(* Logix 5000 project; controller reports 1756-L63 rev 20.11; software revision 20.04; part 17 of 52 *)

        [888].time.Minute := 24, [888].time.Second := 59, [889].log_data[0].min := 1.0, [889].log_data[0].max := 1.0, [889].log_data[0].total := 300.0, [889].log_data[0].time := 300.0, [889].log_data[0].minminute := 25, [889].log_data[0].maxminute := 25, [889].log_data[0].valid := 1, [889].log_data[1].valid := 1, [889].log_data[2].valid := 1, [889].log_data[3].valid := 1, [889].log_data[4].valid := 1, [889].log_data[5].valid := 1, [889].log_data[6].valid := 1, [889].log_data[7].valid := 1, [889].log_data[8].valid := 1, [889].log_data[9].valid := 1, [889].log_data[10].valid := 1, [889].log_data[11].valid := 1, [889].log_data[12].valid := 1, [889].log_data[13].valid := 1, [889].log_data[14].valid := 1, [889].log_data[15].valid := 1, [889].log_data[16].valid := 1, [889].log_data[17].valid := 1, [889].log_data[18].valid := 1, [889].log_data[19].valid := 1, [889].time.Year := 2023, [889].time.Month := 1, [889].time.Day := 12, [889].time.Hour := 18, [889].time.Minute := 29, [889].time.Second := 59, [890].log_data[0].min := 1.0, [890].log_data[0].max := 1.0, [890].log_data[0].total := 300.0, [890].log_data[0].time := 300.0, [890].log_data[0].minminute := 30, [890].log_data[0].maxminute := 30, [890].log_data[0].valid := 1, [890].log_data[1].valid := 1, [890].log_data[2].valid := 1, [890].log_data[3].valid := 1, [890].log_data[4].valid := 1, [890].log_data[5].valid := 1, [890].log_data[6].valid := 1, [890].log_data[7].valid := 1, [890].log_data[8].valid := 1, [890].log_data[9].valid := 1, [890].log_data[10].valid := 1, [890].log_data[11].valid := 1, [890].log_data[12].valid := 1, [890].log_data[13].valid := 1, [890].log_data[14].valid := 1, [890].log_data[15].valid := 1, [890].log_data[16].valid := 1, [890].log_data[17].valid := 1, [890].log_data[18].valid := 1, [890].log_data[19].valid := 1,
        [890].time.Year := 2023, [890].time.Month := 1, [890].time.Day := 12, [890].time.Hour := 18, [890].time.Minute := 34, [890].time.Second := 59, [891].log_data[0].min := 1.0, [891].log_data[0].max := 1.0, [891].log_data[0].total := 300.0, [891].log_data[0].time := 300.0, [891].log_data[0].minminute := 35, [891].log_data[0].maxminute := 35, [891].log_data[0].valid := 1, [891].log_data[1].valid := 1, [891].log_data[2].valid := 1, [891].log_data[3].valid := 1, [891].log_data[4].valid := 1, [891].log_data[5].valid := 1, [891].log_data[6].valid := 1, [891].log_data[7].valid := 1, [891].log_data[8].valid := 1, [891].log_data[9].valid := 1, [891].log_data[10].valid := 1, [891].log_data[11].valid := 1, [891].log_data[12].valid := 1, [891].log_data[13].valid := 1, [891].log_data[14].valid := 1, [891].log_data[15].valid := 1, [891].log_data[16].valid := 1, [891].log_data[17].valid := 1, [891].log_data[18].valid := 1, [891].log_data[19].valid := 1, [891].time.Year := 2023, [891].time.Month := 1, [891].time.Day := 12, [891].time.Hour := 18, [891].time.Minute := 39, [891].time.Second := 59, [892].log_data[0].min := 1.0, [892].log_data[0].max := 1.0, [892].log_data[0].total := 300.0, [892].log_data[0].time := 300.0, [892].log_data[0].minminute := 40, [892].log_data[0].maxminute := 40, [892].log_data[0].valid := 1, [892].log_data[1].valid := 1, [892].log_data[2].valid := 1, [892].log_data[3].valid := 1, [892].log_data[4].valid := 1, [892].log_data[5].valid := 1, [892].log_data[6].valid := 1, [892].log_data[7].valid := 1, [892].log_data[8].valid := 1, [892].log_data[9].valid := 1, [892].log_data[10].valid := 1, [892].log_data[11].valid := 1, [892].log_data[12].valid := 1, [892].log_data[13].valid := 1, [892].log_data[14].valid := 1, [892].log_data[15].valid := 1,
        [892].log_data[16].valid := 1, [892].log_data[17].valid := 1, [892].log_data[18].valid := 1, [892].log_data[19].valid := 1, [892].time.Year := 2023, [892].time.Month := 1, [892].time.Day := 12, [892].time.Hour := 18, [892].time.Minute := 44, [892].time.Second := 59, [893].log_data[0].min := 1.0, [893].log_data[0].max := 1.0, [893].log_data[0].total := 300.0, [893].log_data[0].time := 300.0, [893].log_data[0].minminute := 45, [893].log_data[0].maxminute := 45, [893].log_data[0].valid := 1, [893].log_data[1].valid := 1, [893].log_data[2].valid := 1, [893].log_data[3].valid := 1, [893].log_data[4].valid := 1, [893].log_data[5].valid := 1, [893].log_data[6].valid := 1, [893].log_data[7].valid := 1, [893].log_data[8].valid := 1, [893].log_data[9].valid := 1, [893].log_data[10].valid := 1, [893].log_data[11].valid := 1, [893].log_data[12].valid := 1, [893].log_data[13].valid := 1, [893].log_data[14].valid := 1, [893].log_data[15].valid := 1, [893].log_data[16].valid := 1, [893].log_data[17].valid := 1, [893].log_data[18].valid := 1, [893].log_data[19].valid := 1, [893].time.Year := 2023, [893].time.Month := 1, [893].time.Day := 12, [893].time.Hour := 18, [893].time.Minute := 49, [893].time.Second := 59, [894].log_data[0].min := 1.0, [894].log_data[0].max := 1.0, [894].log_data[0].total := 300.0, [894].log_data[0].time := 300.0, [894].log_data[0].minminute := 50, [894].log_data[0].maxminute := 50, [894].log_data[0].valid := 1, [894].log_data[1].valid := 1, [894].log_data[2].valid := 1, [894].log_data[3].valid := 1, [894].log_data[4].valid := 1, [894].log_data[5].valid := 1, [894].log_data[6].valid := 1, [894].log_data[7].valid := 1, [894].log_data[8].valid := 1, [894].log_data[9].valid := 1, [894].log_data[10].valid := 1, [894].log_data[11].valid := 1,
        [894].log_data[12].valid := 1, [894].log_data[13].valid := 1, [894].log_data[14].valid := 1, [894].log_data[15].valid := 1, [894].log_data[16].valid := 1, [894].log_data[17].valid := 1, [894].log_data[18].valid := 1, [894].log_data[19].valid := 1, [894].time.Year := 2023, [894].time.Month := 1, [894].time.Day := 12, [894].time.Hour := 18, [894].time.Minute := 54, [894].time.Second := 59, [895].log_data[0].min := 1.0, [895].log_data[0].max := 1.0, [895].log_data[0].total := 300.0, [895].log_data[0].time := 300.0, [895].log_data[0].minminute := 55, [895].log_data[0].maxminute := 55, [895].log_data[0].valid := 1, [895].log_data[1].valid := 1, [895].log_data[2].valid := 1, [895].log_data[3].valid := 1, [895].log_data[4].valid := 1, [895].log_data[5].valid := 1, [895].log_data[6].valid := 1, [895].log_data[7].valid := 1, [895].log_data[8].valid := 1, [895].log_data[9].valid := 1, [895].log_data[10].valid := 1, [895].log_data[11].valid := 1, [895].log_data[12].valid := 1, [895].log_data[13].valid := 1, [895].log_data[14].valid := 1, [895].log_data[15].valid := 1, [895].log_data[16].valid := 1, [895].log_data[17].valid := 1, [895].log_data[18].valid := 1, [895].log_data[19].valid := 1, [895].time.Year := 2023, [895].time.Month := 1, [895].time.Day := 12, [895].time.Hour := 18, [895].time.Minute := 59, [895].time.Second := 59, [896].log_data[0].min := 1.0, [896].log_data[0].max := 1.0, [896].log_data[0].total := 300.0, [896].log_data[0].time := 300.0, [896].log_data[0].valid := 1, [896].log_data[1].valid := 1, [896].log_data[2].valid := 1, [896].log_data[3].valid := 1, [896].log_data[4].valid := 1, [896].log_data[5].valid := 1, [896].log_data[6].valid := 1, [896].log_data[7].valid := 1, [896].log_data[8].valid := 1, [896].log_data[9].valid := 1,
        [896].log_data[10].valid := 1, [896].log_data[11].valid := 1, [896].log_data[12].valid := 1, [896].log_data[13].valid := 1, [896].log_data[14].valid := 1, [896].log_data[15].valid := 1, [896].log_data[16].valid := 1, [896].log_data[17].valid := 1, [896].log_data[18].valid := 1, [896].log_data[19].valid := 1, [896].time.Year := 2023, [896].time.Month := 1, [896].time.Day := 12, [896].time.Hour := 19, [896].time.Minute := 4, [896].time.Second := 59, [897].log_data[0].min := 1.0, [897].log_data[0].max := 1.0, [897].log_data[0].total := 300.0, [897].log_data[0].time := 300.0, [897].log_data[0].minminute := 5, [897].log_data[0].maxminute := 5, [897].log_data[0].valid := 1, [897].log_data[1].valid := 1, [897].log_data[2].valid := 1, [897].log_data[3].valid := 1, [897].log_data[4].valid := 1, [897].log_data[5].valid := 1, [897].log_data[6].valid := 1, [897].log_data[7].valid := 1, [897].log_data[8].valid := 1, [897].log_data[9].valid := 1, [897].log_data[10].valid := 1, [897].log_data[11].valid := 1, [897].log_data[12].valid := 1, [897].log_data[13].valid := 1, [897].log_data[14].valid := 1, [897].log_data[15].valid := 1, [897].log_data[16].valid := 1, [897].log_data[17].valid := 1, [897].log_data[18].valid := 1, [897].log_data[19].valid := 1, [897].time.Year := 2023, [897].time.Month := 1, [897].time.Day := 12, [897].time.Hour := 19, [897].time.Minute := 9, [897].time.Second := 59, [898].log_data[0].min := 1.0, [898].log_data[0].max := 1.0, [898].log_data[0].total := 300.0, [898].log_data[0].time := 300.0, [898].log_data[0].minminute := 10, [898].log_data[0].maxminute := 10, [898].log_data[0].valid := 1, [898].log_data[1].valid := 1, [898].log_data[2].valid := 1, [898].log_data[3].valid := 1, [898].log_data[4].valid := 1, [898].log_data[5].valid := 1,
        [898].log_data[6].valid := 1, [898].log_data[7].valid := 1, [898].log_data[8].valid := 1, [898].log_data[9].valid := 1, [898].log_data[10].valid := 1, [898].log_data[11].valid := 1, [898].log_data[12].valid := 1, [898].log_data[13].valid := 1, [898].log_data[14].valid := 1, [898].log_data[15].valid := 1, [898].log_data[16].valid := 1, [898].log_data[17].valid := 1, [898].log_data[18].valid := 1, [898].log_data[19].valid := 1, [898].time.Year := 2023, [898].time.Month := 1, [898].time.Day := 12, [898].time.Hour := 19, [898].time.Minute := 14, [898].time.Second := 59, [899].log_data[0].min := 1.0, [899].log_data[0].max := 1.0, [899].log_data[0].total := 300.0, [899].log_data[0].time := 300.0, [899].log_data[0].minminute := 15, [899].log_data[0].maxminute := 15, [899].log_data[0].valid := 1, [899].log_data[1].valid := 1, [899].log_data[2].valid := 1, [899].log_data[3].valid := 1, [899].log_data[4].valid := 1, [899].log_data[5].valid := 1, [899].log_data[6].valid := 1, [899].log_data[7].valid := 1, [899].log_data[8].valid := 1, [899].log_data[9].valid := 1, [899].log_data[10].valid := 1, [899].log_data[11].valid := 1, [899].log_data[12].valid := 1, [899].log_data[13].valid := 1, [899].log_data[14].valid := 1, [899].log_data[15].valid := 1, [899].log_data[16].valid := 1, [899].log_data[17].valid := 1, [899].log_data[18].valid := 1, [899].log_data[19].valid := 1, [899].time.Year := 2023, [899].time.Month := 1, [899].time.Day := 12, [899].time.Hour := 19, [899].time.Minute := 19, [899].time.Second := 59, [900].log_data[0].min := 1.0, [900].log_data[0].max := 1.0, [900].log_data[0].total := 300.0, [900].log_data[0].time := 300.0, [900].log_data[0].minminute := 20, [900].log_data[0].maxminute := 20, [900].log_data[0].valid := 1, [900].log_data[1].valid := 1,
        [900].log_data[2].valid := 1, [900].log_data[3].valid := 1, [900].log_data[4].valid := 1, [900].log_data[5].valid := 1, [900].log_data[6].valid := 1, [900].log_data[7].valid := 1, [900].log_data[8].valid := 1, [900].log_data[9].valid := 1, [900].log_data[10].valid := 1, [900].log_data[11].valid := 1, [900].log_data[12].valid := 1, [900].log_data[13].valid := 1, [900].log_data[14].valid := 1, [900].log_data[15].valid := 1, [900].log_data[16].valid := 1, [900].log_data[17].valid := 1, [900].log_data[18].valid := 1, [900].log_data[19].valid := 1, [900].time.Year := 2023, [900].time.Month := 1, [900].time.Day := 12, [900].time.Hour := 19, [900].time.Minute := 24, [900].time.Second := 59, [901].log_data[0].min := 1.0, [901].log_data[0].max := 1.0, [901].log_data[0].total := 300.0, [901].log_data[0].time := 300.0, [901].log_data[0].minminute := 25, [901].log_data[0].maxminute := 25, [901].log_data[0].valid := 1, [901].log_data[1].valid := 1, [901].log_data[2].valid := 1, [901].log_data[3].valid := 1, [901].log_data[4].valid := 1, [901].log_data[5].valid := 1, [901].log_data[6].valid := 1, [901].log_data[7].valid := 1, [901].log_data[8].valid := 1, [901].log_data[9].valid := 1, [901].log_data[10].valid := 1, [901].log_data[11].valid := 1, [901].log_data[12].valid := 1, [901].log_data[13].valid := 1, [901].log_data[14].valid := 1, [901].log_data[15].valid := 1, [901].log_data[16].valid := 1, [901].log_data[17].valid := 1, [901].log_data[18].valid := 1, [901].log_data[19].valid := 1, [901].time.Year := 2023, [901].time.Month := 1, [901].time.Day := 12, [901].time.Hour := 19, [901].time.Minute := 29, [901].time.Second := 59, [902].log_data[0].min := 1.0, [902].log_data[0].max := 1.0, [902].log_data[0].total := 300.0, [902].log_data[0].time := 300.0,
        [902].log_data[0].minminute := 30, [902].log_data[0].maxminute := 30, [902].log_data[0].valid := 1, [902].log_data[1].valid := 1, [902].log_data[2].valid := 1, [902].log_data[3].valid := 1, [902].log_data[4].valid := 1, [902].log_data[5].valid := 1, [902].log_data[6].valid := 1, [902].log_data[7].valid := 1, [902].log_data[8].valid := 1, [902].log_data[9].valid := 1, [902].log_data[10].valid := 1, [902].log_data[11].valid := 1, [902].log_data[12].valid := 1, [902].log_data[13].valid := 1, [902].log_data[14].valid := 1, [902].log_data[15].valid := 1, [902].log_data[16].valid := 1, [902].log_data[17].valid := 1, [902].log_data[18].valid := 1, [902].log_data[19].valid := 1, [902].time.Year := 2023, [902].time.Month := 1, [902].time.Day := 12, [902].time.Hour := 19, [902].time.Minute := 34, [902].time.Second := 59, [903].log_data[0].min := 1.0, [903].log_data[0].max := 1.0, [903].log_data[0].total := 300.0, [903].log_data[0].time := 300.0, [903].log_data[0].minminute := 35, [903].log_data[0].maxminute := 35, [903].log_data[0].valid := 1, [903].log_data[1].valid := 1, [903].log_data[2].valid := 1, [903].log_data[3].valid := 1, [903].log_data[4].valid := 1, [903].log_data[5].valid := 1, [903].log_data[6].valid := 1, [903].log_data[7].valid := 1, [903].log_data[8].valid := 1, [903].log_data[9].valid := 1, [903].log_data[10].valid := 1, [903].log_data[11].valid := 1, [903].log_data[12].valid := 1, [903].log_data[13].valid := 1, [903].log_data[14].valid := 1, [903].log_data[15].valid := 1, [903].log_data[16].valid := 1, [903].log_data[17].valid := 1, [903].log_data[18].valid := 1, [903].log_data[19].valid := 1, [903].time.Year := 2023, [903].time.Month := 1, [903].time.Day := 12, [903].time.Hour := 19, [903].time.Minute := 39, [903].time.Second := 59,
        [904].log_data[0].min := 1.0, [904].log_data[0].max := 1.0, [904].log_data[0].total := 300.0, [904].log_data[0].time := 300.0, [904].log_data[0].minminute := 40, [904].log_data[0].maxminute := 40, [904].log_data[0].valid := 1, [904].log_data[1].valid := 1, [904].log_data[2].valid := 1, [904].log_data[3].valid := 1, [904].log_data[4].valid := 1, [904].log_data[5].valid := 1, [904].log_data[6].valid := 1, [904].log_data[7].valid := 1, [904].log_data[8].valid := 1, [904].log_data[9].valid := 1, [904].log_data[10].valid := 1, [904].log_data[11].valid := 1, [904].log_data[12].valid := 1, [904].log_data[13].valid := 1, [904].log_data[14].valid := 1, [904].log_data[15].valid := 1, [904].log_data[16].valid := 1, [904].log_data[17].valid := 1, [904].log_data[18].valid := 1, [904].log_data[19].valid := 1, [904].time.Year := 2023, [904].time.Month := 1, [904].time.Day := 12, [904].time.Hour := 19, [904].time.Minute := 44, [904].time.Second := 59, [905].log_data[0].min := 1.0, [905].log_data[0].max := 1.0, [905].log_data[0].total := 300.0, [905].log_data[0].time := 300.0, [905].log_data[0].minminute := 45, [905].log_data[0].maxminute := 45, [905].log_data[0].valid := 1, [905].log_data[1].valid := 1, [905].log_data[2].valid := 1, [905].log_data[3].valid := 1, [905].log_data[4].valid := 1, [905].log_data[5].valid := 1, [905].log_data[6].valid := 1, [905].log_data[7].valid := 1, [905].log_data[8].valid := 1, [905].log_data[9].valid := 1, [905].log_data[10].valid := 1, [905].log_data[11].valid := 1, [905].log_data[12].valid := 1, [905].log_data[13].valid := 1, [905].log_data[14].valid := 1, [905].log_data[15].valid := 1, [905].log_data[16].valid := 1, [905].log_data[17].valid := 1, [905].log_data[18].valid := 1, [905].log_data[19].valid := 1, [905].time.Year := 2023, [905].time.Month := 1,
        [905].time.Day := 12, [905].time.Hour := 19, [905].time.Minute := 49, [905].time.Second := 59, [906].log_data[0].min := 1.0, [906].log_data[0].max := 1.0, [906].log_data[0].total := 300.0, [906].log_data[0].time := 300.0, [906].log_data[0].minminute := 50, [906].log_data[0].maxminute := 50, [906].log_data[0].valid := 1, [906].log_data[1].valid := 1, [906].log_data[2].valid := 1, [906].log_data[3].valid := 1, [906].log_data[4].valid := 1, [906].log_data[5].valid := 1, [906].log_data[6].valid := 1, [906].log_data[7].valid := 1, [906].log_data[8].valid := 1, [906].log_data[9].valid := 1, [906].log_data[10].valid := 1, [906].log_data[11].valid := 1, [906].log_data[12].valid := 1, [906].log_data[13].valid := 1, [906].log_data[14].valid := 1, [906].log_data[15].valid := 1, [906].log_data[16].valid := 1, [906].log_data[17].valid := 1, [906].log_data[18].valid := 1, [906].log_data[19].valid := 1, [906].time.Year := 2023, [906].time.Month := 1, [906].time.Day := 12, [906].time.Hour := 19, [906].time.Minute := 54, [906].time.Second := 59, [907].log_data[0].min := 1.0, [907].log_data[0].max := 1.0, [907].log_data[0].total := 300.0, [907].log_data[0].time := 300.0, [907].log_data[0].minminute := 55, [907].log_data[0].maxminute := 55, [907].log_data[0].valid := 1, [907].log_data[1].valid := 1, [907].log_data[2].valid := 1, [907].log_data[3].valid := 1, [907].log_data[4].valid := 1, [907].log_data[5].valid := 1, [907].log_data[6].valid := 1, [907].log_data[7].valid := 1, [907].log_data[8].valid := 1, [907].log_data[9].valid := 1, [907].log_data[10].valid := 1, [907].log_data[11].valid := 1, [907].log_data[12].valid := 1, [907].log_data[13].valid := 1, [907].log_data[14].valid := 1, [907].log_data[15].valid := 1, [907].log_data[16].valid := 1, [907].log_data[17].valid := 1,
        [907].log_data[18].valid := 1, [907].log_data[19].valid := 1, [907].time.Year := 2023, [907].time.Month := 1, [907].time.Day := 12, [907].time.Hour := 19, [907].time.Minute := 59, [907].time.Second := 59, [908].log_data[0].min := 1.0, [908].log_data[0].max := 1.0, [908].log_data[0].total := 300.0, [908].log_data[0].time := 300.0, [908].log_data[0].valid := 1, [908].log_data[1].valid := 1, [908].log_data[2].valid := 1, [908].log_data[3].valid := 1, [908].log_data[4].valid := 1, [908].log_data[5].valid := 1, [908].log_data[6].valid := 1, [908].log_data[7].valid := 1, [908].log_data[8].valid := 1, [908].log_data[9].valid := 1, [908].log_data[10].valid := 1, [908].log_data[11].valid := 1, [908].log_data[12].valid := 1, [908].log_data[13].valid := 1, [908].log_data[14].valid := 1, [908].log_data[15].valid := 1, [908].log_data[16].valid := 1, [908].log_data[17].valid := 1, [908].log_data[18].valid := 1, [908].log_data[19].valid := 1, [908].time.Year := 2023, [908].time.Month := 1, [908].time.Day := 12, [908].time.Hour := 20, [908].time.Minute := 4, [908].time.Second := 59, [909].log_data[0].min := 1.0, [909].log_data[0].max := 1.0, [909].log_data[0].total := 300.0, [909].log_data[0].time := 300.0, [909].log_data[0].minminute := 5, [909].log_data[0].maxminute := 5, [909].log_data[0].valid := 1, [909].log_data[1].valid := 1, [909].log_data[2].valid := 1, [909].log_data[3].valid := 1, [909].log_data[4].valid := 1, [909].log_data[5].valid := 1, [909].log_data[6].valid := 1, [909].log_data[7].valid := 1, [909].log_data[8].valid := 1, [909].log_data[9].valid := 1, [909].log_data[10].valid := 1, [909].log_data[11].valid := 1, [909].log_data[12].valid := 1, [909].log_data[13].valid := 1, [909].log_data[14].valid := 1, [909].log_data[15].valid := 1,
        [909].log_data[16].valid := 1, [909].log_data[17].valid := 1, [909].log_data[18].valid := 1, [909].log_data[19].valid := 1, [909].time.Year := 2023, [909].time.Month := 1, [909].time.Day := 12, [909].time.Hour := 20, [909].time.Minute := 9, [909].time.Second := 59, [910].log_data[0].min := 1.0, [910].log_data[0].max := 1.0, [910].log_data[0].total := 300.0, [910].log_data[0].time := 300.0, [910].log_data[0].minminute := 10, [910].log_data[0].maxminute := 10, [910].log_data[0].valid := 1, [910].log_data[1].valid := 1, [910].log_data[2].valid := 1, [910].log_data[3].valid := 1, [910].log_data[4].valid := 1, [910].log_data[5].valid := 1, [910].log_data[6].valid := 1, [910].log_data[7].valid := 1, [910].log_data[8].valid := 1, [910].log_data[9].valid := 1, [910].log_data[10].valid := 1, [910].log_data[11].valid := 1, [910].log_data[12].valid := 1, [910].log_data[13].valid := 1, [910].log_data[14].valid := 1, [910].log_data[15].valid := 1, [910].log_data[16].valid := 1, [910].log_data[17].valid := 1, [910].log_data[18].valid := 1, [910].log_data[19].valid := 1, [910].time.Year := 2023, [910].time.Month := 1, [910].time.Day := 12, [910].time.Hour := 20, [910].time.Minute := 14, [910].time.Second := 59, [911].log_data[0].min := 1.0, [911].log_data[0].max := 1.0, [911].log_data[0].total := 300.0, [911].log_data[0].time := 300.0, [911].log_data[0].minminute := 15, [911].log_data[0].maxminute := 15, [911].log_data[0].valid := 1, [911].log_data[1].valid := 1, [911].log_data[2].valid := 1, [911].log_data[3].valid := 1, [911].log_data[4].valid := 1, [911].log_data[5].valid := 1, [911].log_data[6].valid := 1, [911].log_data[7].valid := 1, [911].log_data[8].valid := 1, [911].log_data[9].valid := 1, [911].log_data[10].valid := 1, [911].log_data[11].valid := 1,
        [911].log_data[12].valid := 1, [911].log_data[13].valid := 1, [911].log_data[14].valid := 1, [911].log_data[15].valid := 1, [911].log_data[16].valid := 1, [911].log_data[17].valid := 1, [911].log_data[18].valid := 1, [911].log_data[19].valid := 1, [911].time.Year := 2023, [911].time.Month := 1, [911].time.Day := 12, [911].time.Hour := 20, [911].time.Minute := 19, [911].time.Second := 59, [912].log_data[0].min := 1.0, [912].log_data[0].max := 1.0, [912].log_data[0].total := 300.0, [912].log_data[0].time := 300.0, [912].log_data[0].minminute := 20, [912].log_data[0].maxminute := 20, [912].log_data[0].valid := 1, [912].log_data[1].valid := 1, [912].log_data[2].valid := 1, [912].log_data[3].valid := 1, [912].log_data[4].valid := 1, [912].log_data[5].valid := 1, [912].log_data[6].valid := 1, [912].log_data[7].valid := 1, [912].log_data[8].valid := 1, [912].log_data[9].valid := 1, [912].log_data[10].valid := 1, [912].log_data[11].valid := 1, [912].log_data[12].valid := 1, [912].log_data[13].valid := 1, [912].log_data[14].valid := 1, [912].log_data[15].valid := 1, [912].log_data[16].valid := 1, [912].log_data[17].valid := 1, [912].log_data[18].valid := 1, [912].log_data[19].valid := 1, [912].time.Year := 2023, [912].time.Month := 1, [912].time.Day := 12, [912].time.Hour := 20, [912].time.Minute := 24, [912].time.Second := 59, [913].log_data[0].min := 1.0, [913].log_data[0].max := 1.0, [913].log_data[0].total := 300.0, [913].log_data[0].time := 300.0, [913].log_data[0].minminute := 25, [913].log_data[0].maxminute := 25, [913].log_data[0].valid := 1, [913].log_data[1].valid := 1, [913].log_data[2].valid := 1, [913].log_data[3].valid := 1, [913].log_data[4].valid := 1, [913].log_data[5].valid := 1, [913].log_data[6].valid := 1, [913].log_data[7].valid := 1,
        [913].log_data[8].valid := 1, [913].log_data[9].valid := 1, [913].log_data[10].valid := 1, [913].log_data[11].valid := 1, [913].log_data[12].valid := 1, [913].log_data[13].valid := 1, [913].log_data[14].valid := 1, [913].log_data[15].valid := 1, [913].log_data[16].valid := 1, [913].log_data[17].valid := 1, [913].log_data[18].valid := 1, [913].log_data[19].valid := 1, [913].time.Year := 2023, [913].time.Month := 1, [913].time.Day := 12, [913].time.Hour := 20, [913].time.Minute := 29, [913].time.Second := 59, [914].log_data[0].min := 1.0, [914].log_data[0].max := 1.0, [914].log_data[0].total := 300.0, [914].log_data[0].time := 300.0, [914].log_data[0].minminute := 30, [914].log_data[0].maxminute := 30, [914].log_data[0].valid := 1, [914].log_data[1].valid := 1, [914].log_data[2].valid := 1, [914].log_data[3].valid := 1, [914].log_data[4].valid := 1, [914].log_data[5].valid := 1, [914].log_data[6].valid := 1, [914].log_data[7].valid := 1, [914].log_data[8].valid := 1, [914].log_data[9].valid := 1, [914].log_data[10].valid := 1, [914].log_data[11].valid := 1, [914].log_data[12].valid := 1, [914].log_data[13].valid := 1, [914].log_data[14].valid := 1, [914].log_data[15].valid := 1, [914].log_data[16].valid := 1, [914].log_data[17].valid := 1, [914].log_data[18].valid := 1, [914].log_data[19].valid := 1, [914].time.Year := 2023, [914].time.Month := 1, [914].time.Day := 12, [914].time.Hour := 20, [914].time.Minute := 34, [914].time.Second := 59, [915].log_data[0].min := 1.0, [915].log_data[0].max := 1.0, [915].log_data[0].total := 300.0, [915].log_data[0].time := 300.0, [915].log_data[0].minminute := 35, [915].log_data[0].maxminute := 35, [915].log_data[0].valid := 1, [915].log_data[1].valid := 1, [915].log_data[2].valid := 1, [915].log_data[3].valid := 1,
        [915].log_data[4].valid := 1, [915].log_data[5].valid := 1, [915].log_data[6].valid := 1, [915].log_data[7].valid := 1, [915].log_data[8].valid := 1, [915].log_data[9].valid := 1, [915].log_data[10].valid := 1, [915].log_data[11].valid := 1, [915].log_data[12].valid := 1, [915].log_data[13].valid := 1, [915].log_data[14].valid := 1, [915].log_data[15].valid := 1, [915].log_data[16].valid := 1, [915].log_data[17].valid := 1, [915].log_data[18].valid := 1, [915].log_data[19].valid := 1, [915].time.Year := 2023, [915].time.Month := 1, [915].time.Day := 12, [915].time.Hour := 20, [915].time.Minute := 39, [915].time.Second := 59, [916].log_data[0].min := 1.0, [916].log_data[0].max := 1.0, [916].log_data[0].total := 300.0, [916].log_data[0].time := 300.0, [916].log_data[0].minminute := 40, [916].log_data[0].maxminute := 40, [916].log_data[0].valid := 1, [916].log_data[1].valid := 1, [916].log_data[2].valid := 1, [916].log_data[3].valid := 1, [916].log_data[4].valid := 1, [916].log_data[5].valid := 1, [916].log_data[6].valid := 1, [916].log_data[7].valid := 1, [916].log_data[8].valid := 1, [916].log_data[9].valid := 1, [916].log_data[10].valid := 1, [916].log_data[11].valid := 1, [916].log_data[12].valid := 1, [916].log_data[13].valid := 1, [916].log_data[14].valid := 1, [916].log_data[15].valid := 1, [916].log_data[16].valid := 1, [916].log_data[17].valid := 1, [916].log_data[18].valid := 1, [916].log_data[19].valid := 1, [916].time.Year := 2023, [916].time.Month := 1, [916].time.Day := 12, [916].time.Hour := 20, [916].time.Minute := 44, [916].time.Second := 59, [917].log_data[0].min := 1.0, [917].log_data[0].max := 1.0, [917].log_data[0].total := 300.0, [917].log_data[0].time := 300.0, [917].log_data[0].minminute := 45, [917].log_data[0].maxminute := 45,
        [917].log_data[0].valid := 1, [917].log_data[1].valid := 1, [917].log_data[2].valid := 1, [917].log_data[3].valid := 1, [917].log_data[4].valid := 1, [917].log_data[5].valid := 1, [917].log_data[6].valid := 1, [917].log_data[7].valid := 1, [917].log_data[8].valid := 1, [917].log_data[9].valid := 1, [917].log_data[10].valid := 1, [917].log_data[11].valid := 1, [917].log_data[12].valid := 1, [917].log_data[13].valid := 1, [917].log_data[14].valid := 1, [917].log_data[15].valid := 1, [917].log_data[16].valid := 1, [917].log_data[17].valid := 1, [917].log_data[18].valid := 1, [917].log_data[19].valid := 1, [917].time.Year := 2023, [917].time.Month := 1, [917].time.Day := 12, [917].time.Hour := 20, [917].time.Minute := 49, [917].time.Second := 59, [918].log_data[0].min := 1.0, [918].log_data[0].max := 1.0, [918].log_data[0].total := 300.0, [918].log_data[0].time := 300.0, [918].log_data[0].minminute := 50, [918].log_data[0].maxminute := 50, [918].log_data[0].valid := 1, [918].log_data[1].valid := 1, [918].log_data[2].valid := 1, [918].log_data[3].valid := 1, [918].log_data[4].valid := 1, [918].log_data[5].valid := 1, [918].log_data[6].valid := 1, [918].log_data[7].valid := 1, [918].log_data[8].valid := 1, [918].log_data[9].valid := 1, [918].log_data[10].valid := 1, [918].log_data[11].valid := 1, [918].log_data[12].valid := 1, [918].log_data[13].valid := 1, [918].log_data[14].valid := 1, [918].log_data[15].valid := 1, [918].log_data[16].valid := 1, [918].log_data[17].valid := 1, [918].log_data[18].valid := 1, [918].log_data[19].valid := 1, [918].time.Year := 2023, [918].time.Month := 1, [918].time.Day := 12, [918].time.Hour := 20, [918].time.Minute := 54, [918].time.Second := 59, [919].log_data[0].min := 1.0, [919].log_data[0].max := 1.0,
        [919].log_data[0].total := 300.0, [919].log_data[0].time := 300.0, [919].log_data[0].minminute := 55, [919].log_data[0].maxminute := 55, [919].log_data[0].valid := 1, [919].log_data[1].valid := 1, [919].log_data[2].valid := 1, [919].log_data[3].valid := 1, [919].log_data[4].valid := 1, [919].log_data[5].valid := 1, [919].log_data[6].valid := 1, [919].log_data[7].valid := 1, [919].log_data[8].valid := 1, [919].log_data[9].valid := 1, [919].log_data[10].valid := 1, [919].log_data[11].valid := 1, [919].log_data[12].valid := 1, [919].log_data[13].valid := 1, [919].log_data[14].valid := 1, [919].log_data[15].valid := 1, [919].log_data[16].valid := 1, [919].log_data[17].valid := 1, [919].log_data[18].valid := 1, [919].log_data[19].valid := 1, [919].time.Year := 2023, [919].time.Month := 1, [919].time.Day := 12, [919].time.Hour := 20, [919].time.Minute := 59, [919].time.Second := 59, [920].log_data[0].min := 1.0, [920].log_data[0].max := 1.0, [920].log_data[0].total := 300.0, [920].log_data[0].time := 300.0, [920].log_data[0].valid := 1, [920].log_data[1].valid := 1, [920].log_data[2].valid := 1, [920].log_data[3].valid := 1, [920].log_data[4].valid := 1, [920].log_data[5].valid := 1, [920].log_data[6].valid := 1, [920].log_data[7].valid := 1, [920].log_data[8].valid := 1, [920].log_data[9].valid := 1, [920].log_data[10].valid := 1, [920].log_data[11].valid := 1, [920].log_data[12].valid := 1, [920].log_data[13].valid := 1, [920].log_data[14].valid := 1, [920].log_data[15].valid := 1, [920].log_data[16].valid := 1, [920].log_data[17].valid := 1, [920].log_data[18].valid := 1, [920].log_data[19].valid := 1, [920].time.Year := 2023, [920].time.Month := 1, [920].time.Day := 12, [920].time.Hour := 21, [920].time.Minute := 4, [920].time.Second := 59,
        [921].log_data[0].min := 1.0, [921].log_data[0].max := 1.0, [921].log_data[0].total := 300.0, [921].log_data[0].time := 300.0, [921].log_data[0].minminute := 5, [921].log_data[0].maxminute := 5, [921].log_data[0].valid := 1, [921].log_data[1].valid := 1, [921].log_data[2].valid := 1, [921].log_data[3].valid := 1, [921].log_data[4].valid := 1, [921].log_data[5].valid := 1, [921].log_data[6].valid := 1, [921].log_data[7].valid := 1, [921].log_data[8].valid := 1, [921].log_data[9].valid := 1, [921].log_data[10].valid := 1, [921].log_data[11].valid := 1, [921].log_data[12].valid := 1, [921].log_data[13].valid := 1, [921].log_data[14].valid := 1, [921].log_data[15].valid := 1, [921].log_data[16].valid := 1, [921].log_data[17].valid := 1, [921].log_data[18].valid := 1, [921].log_data[19].valid := 1, [921].time.Year := 2023, [921].time.Month := 1, [921].time.Day := 12, [921].time.Hour := 21, [921].time.Minute := 9, [921].time.Second := 59, [922].log_data[0].min := 1.0, [922].log_data[0].max := 1.0, [922].log_data[0].total := 300.0, [922].log_data[0].time := 300.0, [922].log_data[0].minminute := 10, [922].log_data[0].maxminute := 10, [922].log_data[0].valid := 1, [922].log_data[1].valid := 1, [922].log_data[2].valid := 1, [922].log_data[3].valid := 1, [922].log_data[4].valid := 1, [922].log_data[5].valid := 1, [922].log_data[6].valid := 1, [922].log_data[7].valid := 1, [922].log_data[8].valid := 1, [922].log_data[9].valid := 1, [922].log_data[10].valid := 1, [922].log_data[11].valid := 1, [922].log_data[12].valid := 1, [922].log_data[13].valid := 1, [922].log_data[14].valid := 1, [922].log_data[15].valid := 1, [922].log_data[16].valid := 1, [922].log_data[17].valid := 1, [922].log_data[18].valid := 1, [922].log_data[19].valid := 1, [922].time.Year := 2023, [922].time.Month := 1,
        [922].time.Day := 12, [922].time.Hour := 21, [922].time.Minute := 14, [922].time.Second := 59, [923].log_data[0].min := 1.0, [923].log_data[0].max := 1.0, [923].log_data[0].total := 300.0, [923].log_data[0].time := 300.0, [923].log_data[0].minminute := 15, [923].log_data[0].maxminute := 15, [923].log_data[0].valid := 1, [923].log_data[1].valid := 1, [923].log_data[2].valid := 1, [923].log_data[3].valid := 1, [923].log_data[4].valid := 1, [923].log_data[5].valid := 1, [923].log_data[6].valid := 1, [923].log_data[7].valid := 1, [923].log_data[8].valid := 1, [923].log_data[9].valid := 1, [923].log_data[10].valid := 1, [923].log_data[11].valid := 1, [923].log_data[12].valid := 1, [923].log_data[13].valid := 1, [923].log_data[14].valid := 1, [923].log_data[15].valid := 1, [923].log_data[16].valid := 1, [923].log_data[17].valid := 1, [923].log_data[18].valid := 1, [923].log_data[19].valid := 1, [923].time.Year := 2023, [923].time.Month := 1, [923].time.Day := 12, [923].time.Hour := 21, [923].time.Minute := 19, [923].time.Second := 59, [924].log_data[0].min := 1.0, [924].log_data[0].max := 1.0, [924].log_data[0].total := 300.0, [924].log_data[0].time := 300.0, [924].log_data[0].minminute := 20, [924].log_data[0].maxminute := 20, [924].log_data[0].valid := 1, [924].log_data[1].valid := 1, [924].log_data[2].valid := 1, [924].log_data[3].valid := 1, [924].log_data[4].valid := 1, [924].log_data[5].valid := 1, [924].log_data[6].valid := 1, [924].log_data[7].valid := 1, [924].log_data[8].valid := 1, [924].log_data[9].valid := 1, [924].log_data[10].valid := 1, [924].log_data[11].valid := 1, [924].log_data[12].valid := 1, [924].log_data[13].valid := 1, [924].log_data[14].valid := 1, [924].log_data[15].valid := 1, [924].log_data[16].valid := 1, [924].log_data[17].valid := 1,
        [924].log_data[18].valid := 1, [924].log_data[19].valid := 1, [924].time.Year := 2023, [924].time.Month := 1, [924].time.Day := 12, [924].time.Hour := 21, [924].time.Minute := 24, [924].time.Second := 59, [925].log_data[0].min := 1.0, [925].log_data[0].max := 1.0, [925].log_data[0].total := 300.0, [925].log_data[0].time := 300.0, [925].log_data[0].minminute := 25, [925].log_data[0].maxminute := 25, [925].log_data[0].valid := 1, [925].log_data[1].valid := 1, [925].log_data[2].valid := 1, [925].log_data[3].valid := 1, [925].log_data[4].valid := 1, [925].log_data[5].valid := 1, [925].log_data[6].valid := 1, [925].log_data[7].valid := 1, [925].log_data[8].valid := 1, [925].log_data[9].valid := 1, [925].log_data[10].valid := 1, [925].log_data[11].valid := 1, [925].log_data[12].valid := 1, [925].log_data[13].valid := 1, [925].log_data[14].valid := 1, [925].log_data[15].valid := 1, [925].log_data[16].valid := 1, [925].log_data[17].valid := 1, [925].log_data[18].valid := 1, [925].log_data[19].valid := 1, [925].time.Year := 2023, [925].time.Month := 1, [925].time.Day := 12, [925].time.Hour := 21, [925].time.Minute := 29, [925].time.Second := 59, [926].log_data[0].min := 1.0, [926].log_data[0].max := 1.0, [926].log_data[0].total := 300.0, [926].log_data[0].time := 300.0, [926].log_data[0].minminute := 30, [926].log_data[0].maxminute := 30, [926].log_data[0].valid := 1, [926].log_data[1].valid := 1, [926].log_data[2].valid := 1, [926].log_data[3].valid := 1, [926].log_data[4].valid := 1, [926].log_data[5].valid := 1, [926].log_data[6].valid := 1, [926].log_data[7].valid := 1, [926].log_data[8].valid := 1, [926].log_data[9].valid := 1, [926].log_data[10].valid := 1, [926].log_data[11].valid := 1, [926].log_data[12].valid := 1, [926].log_data[13].valid := 1,
        [926].log_data[14].valid := 1, [926].log_data[15].valid := 1, [926].log_data[16].valid := 1, [926].log_data[17].valid := 1, [926].log_data[18].valid := 1, [926].log_data[19].valid := 1, [926].time.Year := 2023, [926].time.Month := 1, [926].time.Day := 12, [926].time.Hour := 21, [926].time.Minute := 34, [926].time.Second := 59, [927].log_data[0].min := 1.0, [927].log_data[0].max := 1.0, [927].log_data[0].total := 300.0, [927].log_data[0].time := 300.0, [927].log_data[0].minminute := 35, [927].log_data[0].maxminute := 35, [927].log_data[0].valid := 1, [927].log_data[1].valid := 1, [927].log_data[2].valid := 1, [927].log_data[3].valid := 1, [927].log_data[4].valid := 1, [927].log_data[5].valid := 1, [927].log_data[6].valid := 1, [927].log_data[7].valid := 1, [927].log_data[8].valid := 1, [927].log_data[9].valid := 1, [927].log_data[10].valid := 1, [927].log_data[11].valid := 1, [927].log_data[12].valid := 1, [927].log_data[13].valid := 1, [927].log_data[14].valid := 1, [927].log_data[15].valid := 1, [927].log_data[16].valid := 1, [927].log_data[17].valid := 1, [927].log_data[18].valid := 1, [927].log_data[19].valid := 1, [927].time.Year := 2023, [927].time.Month := 1, [927].time.Day := 12, [927].time.Hour := 21, [927].time.Minute := 39, [927].time.Second := 59, [928].log_data[0].min := 1.0, [928].log_data[0].max := 1.0, [928].log_data[0].total := 300.0, [928].log_data[0].time := 300.0, [928].log_data[0].minminute := 40, [928].log_data[0].maxminute := 40, [928].log_data[0].valid := 1, [928].log_data[1].valid := 1, [928].log_data[2].valid := 1, [928].log_data[3].valid := 1, [928].log_data[4].valid := 1, [928].log_data[5].valid := 1, [928].log_data[6].valid := 1, [928].log_data[7].valid := 1, [928].log_data[8].valid := 1, [928].log_data[9].valid := 1,
        [928].log_data[10].valid := 1, [928].log_data[11].valid := 1, [928].log_data[12].valid := 1, [928].log_data[13].valid := 1, [928].log_data[14].valid := 1, [928].log_data[15].valid := 1, [928].log_data[16].valid := 1, [928].log_data[17].valid := 1, [928].log_data[18].valid := 1, [928].log_data[19].valid := 1, [928].time.Year := 2023, [928].time.Month := 1, [928].time.Day := 12, [928].time.Hour := 21, [928].time.Minute := 44, [928].time.Second := 59, [929].log_data[0].min := 1.0, [929].log_data[0].max := 1.0, [929].log_data[0].total := 300.0, [929].log_data[0].time := 300.0, [929].log_data[0].minminute := 45, [929].log_data[0].maxminute := 45, [929].log_data[0].valid := 1, [929].log_data[1].valid := 1, [929].log_data[2].valid := 1, [929].log_data[3].valid := 1, [929].log_data[4].valid := 1, [929].log_data[5].valid := 1, [929].log_data[6].valid := 1, [929].log_data[7].valid := 1, [929].log_data[8].valid := 1, [929].log_data[9].valid := 1, [929].log_data[10].valid := 1, [929].log_data[11].valid := 1, [929].log_data[12].valid := 1, [929].log_data[13].valid := 1, [929].log_data[14].valid := 1, [929].log_data[15].valid := 1, [929].log_data[16].valid := 1, [929].log_data[17].valid := 1, [929].log_data[18].valid := 1, [929].log_data[19].valid := 1, [929].time.Year := 2023, [929].time.Month := 1, [929].time.Day := 12, [929].time.Hour := 21, [929].time.Minute := 49, [929].time.Second := 59, [930].log_data[0].min := 1.0, [930].log_data[0].max := 1.0, [930].log_data[0].total := 300.0, [930].log_data[0].time := 300.0, [930].log_data[0].minminute := 50, [930].log_data[0].maxminute := 50, [930].log_data[0].valid := 1, [930].log_data[1].valid := 1, [930].log_data[2].valid := 1, [930].log_data[3].valid := 1, [930].log_data[4].valid := 1, [930].log_data[5].valid := 1,
        [930].log_data[6].valid := 1, [930].log_data[7].valid := 1, [930].log_data[8].valid := 1, [930].log_data[9].valid := 1, [930].log_data[10].valid := 1, [930].log_data[11].valid := 1, [930].log_data[12].valid := 1, [930].log_data[13].valid := 1, [930].log_data[14].valid := 1, [930].log_data[15].valid := 1, [930].log_data[16].valid := 1, [930].log_data[17].valid := 1, [930].log_data[18].valid := 1, [930].log_data[19].valid := 1, [930].time.Year := 2023, [930].time.Month := 1, [930].time.Day := 12, [930].time.Hour := 21, [930].time.Minute := 54, [930].time.Second := 59, [931].log_data[0].min := 1.0, [931].log_data[0].max := 1.0, [931].log_data[0].total := 300.0, [931].log_data[0].time := 300.0, [931].log_data[0].minminute := 55, [931].log_data[0].maxminute := 55, [931].log_data[0].valid := 1, [931].log_data[1].valid := 1, [931].log_data[2].valid := 1, [931].log_data[3].valid := 1, [931].log_data[4].valid := 1, [931].log_data[5].valid := 1, [931].log_data[6].valid := 1, [931].log_data[7].valid := 1, [931].log_data[8].valid := 1, [931].log_data[9].valid := 1, [931].log_data[10].valid := 1, [931].log_data[11].valid := 1, [931].log_data[12].valid := 1, [931].log_data[13].valid := 1, [931].log_data[14].valid := 1, [931].log_data[15].valid := 1, [931].log_data[16].valid := 1, [931].log_data[17].valid := 1, [931].log_data[18].valid := 1, [931].log_data[19].valid := 1, [931].time.Year := 2023, [931].time.Month := 1, [931].time.Day := 12, [931].time.Hour := 21, [931].time.Minute := 59, [931].time.Second := 59, [932].log_data[0].min := 1.0, [932].log_data[0].max := 1.0, [932].log_data[0].total := 300.0, [932].log_data[0].time := 300.0, [932].log_data[0].valid := 1, [932].log_data[1].valid := 1, [932].log_data[2].valid := 1, [932].log_data[3].valid := 1,
        [932].log_data[4].valid := 1, [932].log_data[5].valid := 1, [932].log_data[6].valid := 1, [932].log_data[7].valid := 1, [932].log_data[8].valid := 1, [932].log_data[9].valid := 1, [932].log_data[10].valid := 1, [932].log_data[11].valid := 1, [932].log_data[12].valid := 1, [932].log_data[13].valid := 1, [932].log_data[14].valid := 1, [932].log_data[15].valid := 1, [932].log_data[16].valid := 1, [932].log_data[17].valid := 1, [932].log_data[18].valid := 1, [932].log_data[19].valid := 1, [932].time.Year := 2023, [932].time.Month := 1, [932].time.Day := 12, [932].time.Hour := 22, [932].time.Minute := 4, [932].time.Second := 59, [933].log_data[0].min := 1.0, [933].log_data[0].max := 1.0, [933].log_data[0].total := 300.0, [933].log_data[0].time := 300.0, [933].log_data[0].minminute := 5, [933].log_data[0].maxminute := 5, [933].log_data[0].valid := 1, [933].log_data[1].valid := 1, [933].log_data[2].valid := 1, [933].log_data[3].valid := 1, [933].log_data[4].valid := 1, [933].log_data[5].valid := 1, [933].log_data[6].valid := 1, [933].log_data[7].valid := 1, [933].log_data[8].valid := 1, [933].log_data[9].valid := 1, [933].log_data[10].valid := 1, [933].log_data[11].valid := 1, [933].log_data[12].valid := 1, [933].log_data[13].valid := 1, [933].log_data[14].valid := 1, [933].log_data[15].valid := 1, [933].log_data[16].valid := 1, [933].log_data[17].valid := 1, [933].log_data[18].valid := 1, [933].log_data[19].valid := 1, [933].time.Year := 2023, [933].time.Month := 1, [933].time.Day := 12, [933].time.Hour := 22, [933].time.Minute := 9, [933].time.Second := 59, [934].log_data[0].min := 1.0, [934].log_data[0].max := 1.0, [934].log_data[0].total := 300.0, [934].log_data[0].time := 300.0, [934].log_data[0].minminute := 10, [934].log_data[0].maxminute := 10,
        [934].log_data[0].valid := 1, [934].log_data[1].valid := 1, [934].log_data[2].valid := 1, [934].log_data[3].valid := 1, [934].log_data[4].valid := 1, [934].log_data[5].valid := 1, [934].log_data[6].valid := 1, [934].log_data[7].valid := 1, [934].log_data[8].valid := 1, [934].log_data[9].valid := 1, [934].log_data[10].valid := 1, [934].log_data[11].valid := 1, [934].log_data[12].valid := 1, [934].log_data[13].valid := 1, [934].log_data[14].valid := 1, [934].log_data[15].valid := 1, [934].log_data[16].valid := 1, [934].log_data[17].valid := 1, [934].log_data[18].valid := 1, [934].log_data[19].valid := 1, [934].time.Year := 2023, [934].time.Month := 1, [934].time.Day := 12, [934].time.Hour := 22, [934].time.Minute := 14, [934].time.Second := 59, [935].log_data[0].min := 1.0, [935].log_data[0].max := 1.0, [935].log_data[0].total := 300.0, [935].log_data[0].time := 300.0, [935].log_data[0].minminute := 15, [935].log_data[0].maxminute := 15, [935].log_data[0].valid := 1, [935].log_data[1].valid := 1, [935].log_data[2].valid := 1, [935].log_data[3].valid := 1, [935].log_data[4].valid := 1, [935].log_data[5].valid := 1, [935].log_data[6].valid := 1, [935].log_data[7].valid := 1, [935].log_data[8].valid := 1, [935].log_data[9].valid := 1, [935].log_data[10].valid := 1, [935].log_data[11].valid := 1, [935].log_data[12].valid := 1, [935].log_data[13].valid := 1, [935].log_data[14].valid := 1, [935].log_data[15].valid := 1, [935].log_data[16].valid := 1, [935].log_data[17].valid := 1, [935].log_data[18].valid := 1, [935].log_data[19].valid := 1, [935].time.Year := 2023, [935].time.Month := 1, [935].time.Day := 12, [935].time.Hour := 22, [935].time.Minute := 19, [935].time.Second := 59, [936].log_data[0].min := 1.0, [936].log_data[0].max := 1.0,
        [936].log_data[0].total := 300.0, [936].log_data[0].time := 300.0, [936].log_data[0].minminute := 20, [936].log_data[0].maxminute := 20, [936].log_data[0].valid := 1, [936].log_data[1].valid := 1, [936].log_data[2].valid := 1, [936].log_data[3].valid := 1, [936].log_data[4].valid := 1, [936].log_data[5].valid := 1, [936].log_data[6].valid := 1, [936].log_data[7].valid := 1, [936].log_data[8].valid := 1, [936].log_data[9].valid := 1, [936].log_data[10].valid := 1, [936].log_data[11].valid := 1, [936].log_data[12].valid := 1, [936].log_data[13].valid := 1, [936].log_data[14].valid := 1, [936].log_data[15].valid := 1, [936].log_data[16].valid := 1, [936].log_data[17].valid := 1, [936].log_data[18].valid := 1, [936].log_data[19].valid := 1, [936].time.Year := 2023, [936].time.Month := 1, [936].time.Day := 12, [936].time.Hour := 22, [936].time.Minute := 24, [936].time.Second := 59, [937].log_data[0].min := 1.0, [937].log_data[0].max := 1.0, [937].log_data[0].total := 300.0, [937].log_data[0].time := 300.0, [937].log_data[0].minminute := 25, [937].log_data[0].maxminute := 25, [937].log_data[0].valid := 1, [937].log_data[1].valid := 1, [937].log_data[2].valid := 1, [937].log_data[3].valid := 1, [937].log_data[4].valid := 1, [937].log_data[5].valid := 1, [937].log_data[6].valid := 1, [937].log_data[7].valid := 1, [937].log_data[8].valid := 1, [937].log_data[9].valid := 1, [937].log_data[10].valid := 1, [937].log_data[11].valid := 1, [937].log_data[12].valid := 1, [937].log_data[13].valid := 1, [937].log_data[14].valid := 1, [937].log_data[15].valid := 1, [937].log_data[16].valid := 1, [937].log_data[17].valid := 1, [937].log_data[18].valid := 1, [937].log_data[19].valid := 1, [937].time.Year := 2023, [937].time.Month := 1, [937].time.Day := 12, [937].time.Hour := 22,
        [937].time.Minute := 29, [937].time.Second := 59, [938].log_data[0].min := 1.0, [938].log_data[0].max := 1.0, [938].log_data[0].total := 300.0, [938].log_data[0].time := 300.0, [938].log_data[0].minminute := 30, [938].log_data[0].maxminute := 30, [938].log_data[0].valid := 1, [938].log_data[1].valid := 1, [938].log_data[2].valid := 1, [938].log_data[3].valid := 1, [938].log_data[4].valid := 1, [938].log_data[5].valid := 1, [938].log_data[6].valid := 1, [938].log_data[7].valid := 1, [938].log_data[8].valid := 1, [938].log_data[9].valid := 1, [938].log_data[10].valid := 1, [938].log_data[11].valid := 1, [938].log_data[12].valid := 1, [938].log_data[13].valid := 1, [938].log_data[14].valid := 1, [938].log_data[15].valid := 1, [938].log_data[16].valid := 1, [938].log_data[17].valid := 1, [938].log_data[18].valid := 1, [938].log_data[19].valid := 1, [938].time.Year := 2023, [938].time.Month := 1, [938].time.Day := 12, [938].time.Hour := 22, [938].time.Minute := 34, [938].time.Second := 59, [939].log_data[0].min := 1.0, [939].log_data[0].max := 1.0, [939].log_data[0].total := 300.0, [939].log_data[0].time := 300.0, [939].log_data[0].minminute := 35, [939].log_data[0].maxminute := 35, [939].log_data[0].valid := 1, [939].log_data[1].valid := 1, [939].log_data[2].valid := 1, [939].log_data[3].valid := 1, [939].log_data[4].valid := 1, [939].log_data[5].valid := 1, [939].log_data[6].valid := 1, [939].log_data[7].valid := 1, [939].log_data[8].valid := 1, [939].log_data[9].valid := 1, [939].log_data[10].valid := 1, [939].log_data[11].valid := 1, [939].log_data[12].valid := 1, [939].log_data[13].valid := 1, [939].log_data[14].valid := 1, [939].log_data[15].valid := 1, [939].log_data[16].valid := 1, [939].log_data[17].valid := 1, [939].log_data[18].valid := 1, [939].log_data[19].valid := 1,
        [939].time.Year := 2023, [939].time.Month := 1, [939].time.Day := 12, [939].time.Hour := 22, [939].time.Minute := 39, [939].time.Second := 59, [940].log_data[0].min := 1.0, [940].log_data[0].max := 1.0, [940].log_data[0].total := 300.0, [940].log_data[0].time := 300.0, [940].log_data[0].minminute := 40, [940].log_data[0].maxminute := 40, [940].log_data[0].valid := 1, [940].log_data[1].valid := 1, [940].log_data[2].valid := 1, [940].log_data[3].valid := 1, [940].log_data[4].valid := 1, [940].log_data[5].valid := 1, [940].log_data[6].valid := 1, [940].log_data[7].valid := 1, [940].log_data[8].valid := 1, [940].log_data[9].valid := 1, [940].log_data[10].valid := 1, [940].log_data[11].valid := 1, [940].log_data[12].valid := 1, [940].log_data[13].valid := 1, [940].log_data[14].valid := 1, [940].log_data[15].valid := 1, [940].log_data[16].valid := 1, [940].log_data[17].valid := 1, [940].log_data[18].valid := 1, [940].log_data[19].valid := 1, [940].time.Year := 2023, [940].time.Month := 1, [940].time.Day := 12, [940].time.Hour := 22, [940].time.Minute := 44, [940].time.Second := 59, [941].log_data[0].min := 1.0, [941].log_data[0].max := 1.0, [941].log_data[0].total := 300.0, [941].log_data[0].time := 300.0, [941].log_data[0].minminute := 45, [941].log_data[0].maxminute := 45, [941].log_data[0].valid := 1, [941].log_data[1].valid := 1, [941].log_data[2].valid := 1, [941].log_data[3].valid := 1, [941].log_data[4].valid := 1, [941].log_data[5].valid := 1, [941].log_data[6].valid := 1, [941].log_data[7].valid := 1, [941].log_data[8].valid := 1, [941].log_data[9].valid := 1, [941].log_data[10].valid := 1, [941].log_data[11].valid := 1, [941].log_data[12].valid := 1, [941].log_data[13].valid := 1, [941].log_data[14].valid := 1, [941].log_data[15].valid := 1,
        [941].log_data[16].valid := 1, [941].log_data[17].valid := 1, [941].log_data[18].valid := 1, [941].log_data[19].valid := 1, [941].time.Year := 2023, [941].time.Month := 1, [941].time.Day := 12, [941].time.Hour := 22, [941].time.Minute := 49, [941].time.Second := 59, [942].log_data[0].min := 1.0, [942].log_data[0].max := 1.0, [942].log_data[0].total := 300.0, [942].log_data[0].time := 300.0, [942].log_data[0].minminute := 50, [942].log_data[0].maxminute := 50, [942].log_data[0].valid := 1, [942].log_data[1].valid := 1, [942].log_data[2].valid := 1, [942].log_data[3].valid := 1, [942].log_data[4].valid := 1, [942].log_data[5].valid := 1, [942].log_data[6].valid := 1, [942].log_data[7].valid := 1, [942].log_data[8].valid := 1, [942].log_data[9].valid := 1, [942].log_data[10].valid := 1, [942].log_data[11].valid := 1, [942].log_data[12].valid := 1, [942].log_data[13].valid := 1, [942].log_data[14].valid := 1, [942].log_data[15].valid := 1, [942].log_data[16].valid := 1, [942].log_data[17].valid := 1, [942].log_data[18].valid := 1, [942].log_data[19].valid := 1, [942].time.Year := 2023, [942].time.Month := 1, [942].time.Day := 12, [942].time.Hour := 22, [942].time.Minute := 54, [942].time.Second := 59, [943].log_data[0].min := 1.0, [943].log_data[0].max := 1.0, [943].log_data[0].total := 300.0, [943].log_data[0].time := 300.0, [943].log_data[0].minminute := 55, [943].log_data[0].maxminute := 55, [943].log_data[0].valid := 1, [943].log_data[1].valid := 1, [943].log_data[2].valid := 1, [943].log_data[3].valid := 1, [943].log_data[4].valid := 1, [943].log_data[5].valid := 1, [943].log_data[6].valid := 1, [943].log_data[7].valid := 1, [943].log_data[8].valid := 1, [943].log_data[9].valid := 1, [943].log_data[10].valid := 1, [943].log_data[11].valid := 1,
        [943].log_data[12].valid := 1, [943].log_data[13].valid := 1, [943].log_data[14].valid := 1, [943].log_data[15].valid := 1, [943].log_data[16].valid := 1, [943].log_data[17].valid := 1, [943].log_data[18].valid := 1, [943].log_data[19].valid := 1, [943].time.Year := 2023, [943].time.Month := 1, [943].time.Day := 12, [943].time.Hour := 22, [943].time.Minute := 59, [943].time.Second := 59, [944].log_data[0].min := 1.0, [944].log_data[0].max := 1.0, [944].log_data[0].total := 300.0, [944].log_data[0].time := 300.0, [944].log_data[0].valid := 1, [944].log_data[1].valid := 1, [944].log_data[2].valid := 1, [944].log_data[3].valid := 1, [944].log_data[4].valid := 1, [944].log_data[5].valid := 1, [944].log_data[6].valid := 1, [944].log_data[7].valid := 1, [944].log_data[8].valid := 1, [944].log_data[9].valid := 1, [944].log_data[10].valid := 1, [944].log_data[11].valid := 1, [944].log_data[12].valid := 1, [944].log_data[13].valid := 1, [944].log_data[14].valid := 1, [944].log_data[15].valid := 1, [944].log_data[16].valid := 1, [944].log_data[17].valid := 1, [944].log_data[18].valid := 1, [944].log_data[19].valid := 1, [944].time.Year := 2023, [944].time.Month := 1, [944].time.Day := 12, [944].time.Hour := 23, [944].time.Minute := 4, [944].time.Second := 59, [945].log_data[0].min := 1.0, [945].log_data[0].max := 1.0, [945].log_data[0].total := 300.0, [945].log_data[0].time := 300.0, [945].log_data[0].minminute := 5, [945].log_data[0].maxminute := 5, [945].log_data[0].valid := 1, [945].log_data[1].valid := 1, [945].log_data[2].valid := 1, [945].log_data[3].valid := 1, [945].log_data[4].valid := 1, [945].log_data[5].valid := 1, [945].log_data[6].valid := 1, [945].log_data[7].valid := 1, [945].log_data[8].valid := 1, [945].log_data[9].valid := 1,
        [945].log_data[10].valid := 1, [945].log_data[11].valid := 1, [945].log_data[12].valid := 1, [945].log_data[13].valid := 1, [945].log_data[14].valid := 1, [945].log_data[15].valid := 1, [945].log_data[16].valid := 1, [945].log_data[17].valid := 1, [945].log_data[18].valid := 1, [945].log_data[19].valid := 1, [945].time.Year := 2023, [945].time.Month := 1, [945].time.Day := 12, [945].time.Hour := 23, [945].time.Minute := 9, [945].time.Second := 59, [946].log_data[0].min := 1.0, [946].log_data[0].max := 1.0, [946].log_data[0].total := 300.0, [946].log_data[0].time := 300.0, [946].log_data[0].minminute := 10, [946].log_data[0].maxminute := 10, [946].log_data[0].valid := 1, [946].log_data[1].valid := 1, [946].log_data[2].valid := 1, [946].log_data[3].valid := 1, [946].log_data[4].valid := 1, [946].log_data[5].valid := 1, [946].log_data[6].valid := 1, [946].log_data[7].valid := 1, [946].log_data[8].valid := 1, [946].log_data[9].valid := 1, [946].log_data[10].valid := 1, [946].log_data[11].valid := 1, [946].log_data[12].valid := 1, [946].log_data[13].valid := 1, [946].log_data[14].valid := 1, [946].log_data[15].valid := 1, [946].log_data[16].valid := 1, [946].log_data[17].valid := 1, [946].log_data[18].valid := 1, [946].log_data[19].valid := 1, [946].time.Year := 2023, [946].time.Month := 1, [946].time.Day := 12, [946].time.Hour := 23, [946].time.Minute := 14, [946].time.Second := 59, [947].log_data[0].min := 1.0, [947].log_data[0].max := 1.0, [947].log_data[0].total := 300.0, [947].log_data[0].time := 300.0, [947].log_data[0].minminute := 15, [947].log_data[0].maxminute := 15, [947].log_data[0].valid := 1, [947].log_data[1].valid := 1, [947].log_data[2].valid := 1, [947].log_data[3].valid := 1, [947].log_data[4].valid := 1, [947].log_data[5].valid := 1,
        [947].log_data[6].valid := 1, [947].log_data[7].valid := 1, [947].log_data[8].valid := 1, [947].log_data[9].valid := 1, [947].log_data[10].valid := 1, [947].log_data[11].valid := 1, [947].log_data[12].valid := 1, [947].log_data[13].valid := 1, [947].log_data[14].valid := 1, [947].log_data[15].valid := 1, [947].log_data[16].valid := 1, [947].log_data[17].valid := 1, [947].log_data[18].valid := 1, [947].log_data[19].valid := 1, [947].time.Year := 2023, [947].time.Month := 1, [947].time.Day := 12, [947].time.Hour := 23, [947].time.Minute := 19, [947].time.Second := 59, [948].log_data[0].min := 1.0, [948].log_data[0].max := 1.0, [948].log_data[0].total := 300.0, [948].log_data[0].time := 300.0, [948].log_data[0].minminute := 20, [948].log_data[0].maxminute := 20, [948].log_data[0].valid := 1, [948].log_data[1].valid := 1, [948].log_data[2].valid := 1, [948].log_data[3].valid := 1, [948].log_data[4].valid := 1, [948].log_data[5].valid := 1, [948].log_data[6].valid := 1, [948].log_data[7].valid := 1, [948].log_data[8].valid := 1, [948].log_data[9].valid := 1, [948].log_data[10].valid := 1, [948].log_data[11].valid := 1, [948].log_data[12].valid := 1, [948].log_data[13].valid := 1, [948].log_data[14].valid := 1, [948].log_data[15].valid := 1, [948].log_data[16].valid := 1, [948].log_data[17].valid := 1, [948].log_data[18].valid := 1, [948].log_data[19].valid := 1, [948].time.Year := 2023, [948].time.Month := 1, [948].time.Day := 12, [948].time.Hour := 23, [948].time.Minute := 24, [948].time.Second := 59, [949].log_data[0].min := 1.0, [949].log_data[0].max := 1.0, [949].log_data[0].total := 300.0, [949].log_data[0].time := 300.0, [949].log_data[0].minminute := 25, [949].log_data[0].maxminute := 25, [949].log_data[0].valid := 1, [949].log_data[1].valid := 1,
        [949].log_data[2].valid := 1, [949].log_data[3].valid := 1, [949].log_data[4].valid := 1, [949].log_data[5].valid := 1, [949].log_data[6].valid := 1, [949].log_data[7].valid := 1, [949].log_data[8].valid := 1, [949].log_data[9].valid := 1, [949].log_data[10].valid := 1, [949].log_data[11].valid := 1, [949].log_data[12].valid := 1, [949].log_data[13].valid := 1, [949].log_data[14].valid := 1, [949].log_data[15].valid := 1, [949].log_data[16].valid := 1, [949].log_data[17].valid := 1, [949].log_data[18].valid := 1, [949].log_data[19].valid := 1, [949].time.Year := 2023, [949].time.Month := 1, [949].time.Day := 12, [949].time.Hour := 23, [949].time.Minute := 29, [949].time.Second := 59, [950].log_data[0].min := 1.0, [950].log_data[0].max := 1.0, [950].log_data[0].total := 300.0, [950].log_data[0].time := 300.0, [950].log_data[0].minminute := 30, [950].log_data[0].maxminute := 30, [950].log_data[0].valid := 1, [950].log_data[1].valid := 1, [950].log_data[2].valid := 1, [950].log_data[3].valid := 1, [950].log_data[4].valid := 1, [950].log_data[5].valid := 1, [950].log_data[6].valid := 1, [950].log_data[7].valid := 1, [950].log_data[8].valid := 1, [950].log_data[9].valid := 1, [950].log_data[10].valid := 1, [950].log_data[11].valid := 1, [950].log_data[12].valid := 1, [950].log_data[13].valid := 1, [950].log_data[14].valid := 1, [950].log_data[15].valid := 1, [950].log_data[16].valid := 1, [950].log_data[17].valid := 1, [950].log_data[18].valid := 1, [950].log_data[19].valid := 1, [950].time.Year := 2023, [950].time.Month := 1, [950].time.Day := 12, [950].time.Hour := 23, [950].time.Minute := 34, [950].time.Second := 59, [951].log_data[0].min := 1.0, [951].log_data[0].max := 1.0, [951].log_data[0].total := 300.0, [951].log_data[0].time := 300.0,
        [951].log_data[0].minminute := 35, [951].log_data[0].maxminute := 35, [951].log_data[0].valid := 1, [951].log_data[1].valid := 1, [951].log_data[2].valid := 1, [951].log_data[3].valid := 1, [951].log_data[4].valid := 1, [951].log_data[5].valid := 1, [951].log_data[6].valid := 1, [951].log_data[7].valid := 1, [951].log_data[8].valid := 1, [951].log_data[9].valid := 1, [951].log_data[10].valid := 1, [951].log_data[11].valid := 1, [951].log_data[12].valid := 1, [951].log_data[13].valid := 1, [951].log_data[14].valid := 1, [951].log_data[15].valid := 1, [951].log_data[16].valid := 1, [951].log_data[17].valid := 1, [951].log_data[18].valid := 1, [951].log_data[19].valid := 1, [951].time.Year := 2023, [951].time.Month := 1, [951].time.Day := 12, [951].time.Hour := 23, [951].time.Minute := 39, [951].time.Second := 59, [952].log_data[0].min := 1.0, [952].log_data[0].max := 1.0, [952].log_data[0].total := 300.0, [952].log_data[0].time := 300.0, [952].log_data[0].minminute := 40, [952].log_data[0].maxminute := 40, [952].log_data[0].valid := 1, [952].log_data[1].valid := 1, [952].log_data[2].valid := 1, [952].log_data[3].valid := 1, [952].log_data[4].valid := 1, [952].log_data[5].valid := 1, [952].log_data[6].valid := 1, [952].log_data[7].valid := 1, [952].log_data[8].valid := 1, [952].log_data[9].valid := 1, [952].log_data[10].valid := 1, [952].log_data[11].valid := 1, [952].log_data[12].valid := 1, [952].log_data[13].valid := 1, [952].log_data[14].valid := 1, [952].log_data[15].valid := 1, [952].log_data[16].valid := 1, [952].log_data[17].valid := 1, [952].log_data[18].valid := 1, [952].log_data[19].valid := 1, [952].time.Year := 2023, [952].time.Month := 1, [952].time.Day := 12, [952].time.Hour := 23, [952].time.Minute := 44, [952].time.Second := 59,
        [953].log_data[0].min := 1.0, [953].log_data[0].max := 1.0, [953].log_data[0].total := 300.0, [953].log_data[0].time := 300.0, [953].log_data[0].minminute := 45, [953].log_data[0].maxminute := 45, [953].log_data[0].valid := 1, [953].log_data[1].valid := 1, [953].log_data[2].valid := 1, [953].log_data[3].valid := 1, [953].log_data[4].valid := 1, [953].log_data[5].valid := 1, [953].log_data[6].valid := 1, [953].log_data[7].valid := 1, [953].log_data[8].valid := 1, [953].log_data[9].valid := 1, [953].log_data[10].valid := 1, [953].log_data[11].valid := 1, [953].log_data[12].valid := 1, [953].log_data[13].valid := 1, [953].log_data[14].valid := 1, [953].log_data[15].valid := 1, [953].log_data[16].valid := 1, [953].log_data[17].valid := 1, [953].log_data[18].valid := 1, [953].log_data[19].valid := 1, [953].time.Year := 2023, [953].time.Month := 1, [953].time.Day := 12, [953].time.Hour := 23, [953].time.Minute := 49, [953].time.Second := 59, [954].log_data[0].min := 1.0, [954].log_data[0].max := 1.0, [954].log_data[0].total := 300.0, [954].log_data[0].time := 300.0, [954].log_data[0].minminute := 50, [954].log_data[0].maxminute := 50, [954].log_data[0].valid := 1, [954].log_data[1].valid := 1, [954].log_data[2].valid := 1, [954].log_data[3].valid := 1, [954].log_data[4].valid := 1, [954].log_data[5].valid := 1, [954].log_data[6].valid := 1, [954].log_data[7].valid := 1, [954].log_data[8].valid := 1, [954].log_data[9].valid := 1, [954].log_data[10].valid := 1, [954].log_data[11].valid := 1, [954].log_data[12].valid := 1, [954].log_data[13].valid := 1, [954].log_data[14].valid := 1, [954].log_data[15].valid := 1, [954].log_data[16].valid := 1, [954].log_data[17].valid := 1, [954].log_data[18].valid := 1, [954].log_data[19].valid := 1, [954].time.Year := 2023, [954].time.Month := 1,
        [954].time.Day := 12, [954].time.Hour := 23, [954].time.Minute := 54, [954].time.Second := 59, [955].log_data[0].min := 1.0, [955].log_data[0].max := 1.0, [955].log_data[0].total := 300.0, [955].log_data[0].time := 300.0, [955].log_data[0].minminute := 55, [955].log_data[0].maxminute := 55, [955].log_data[0].valid := 1, [955].log_data[1].valid := 1, [955].log_data[2].valid := 1, [955].log_data[3].valid := 1, [955].log_data[4].valid := 1, [955].log_data[5].valid := 1, [955].log_data[6].valid := 1, [955].log_data[7].valid := 1, [955].log_data[8].valid := 1, [955].log_data[9].valid := 1, [955].log_data[10].valid := 1, [955].log_data[11].valid := 1, [955].log_data[12].valid := 1, [955].log_data[13].valid := 1, [955].log_data[14].valid := 1, [955].log_data[15].valid := 1, [955].log_data[16].valid := 1, [955].log_data[17].valid := 1, [955].log_data[18].valid := 1, [955].log_data[19].valid := 1, [955].time.Year := 2023, [955].time.Month := 1, [955].time.Day := 12, [955].time.Hour := 23, [955].time.Minute := 59, [955].time.Second := 59, [956].log_data[0].min := 1.0, [956].log_data[0].max := 1.0, [956].log_data[0].total := 300.0, [956].log_data[0].time := 300.0, [956].log_data[0].valid := 1, [956].log_data[1].valid := 1, [956].log_data[2].valid := 1, [956].log_data[3].valid := 1, [956].log_data[4].valid := 1, [956].log_data[5].valid := 1, [956].log_data[6].valid := 1, [956].log_data[7].valid := 1, [956].log_data[8].valid := 1, [956].log_data[9].valid := 1, [956].log_data[10].valid := 1, [956].log_data[11].valid := 1, [956].log_data[12].valid := 1, [956].log_data[13].valid := 1, [956].log_data[14].valid := 1, [956].log_data[15].valid := 1, [956].log_data[16].valid := 1, [956].log_data[17].valid := 1, [956].log_data[18].valid := 1, [956].log_data[19].valid := 1,
        [956].time.Year := 2023, [956].time.Month := 1, [956].time.Day := 13, [956].time.Minute := 4, [956].time.Second := 59, [957].log_data[0].min := 1.0, [957].log_data[0].max := 1.0, [957].log_data[0].total := 300.0, [957].log_data[0].time := 300.0, [957].log_data[0].minminute := 5, [957].log_data[0].maxminute := 5, [957].log_data[0].valid := 1, [957].log_data[1].valid := 1, [957].log_data[2].valid := 1, [957].log_data[3].valid := 1, [957].log_data[4].valid := 1, [957].log_data[5].valid := 1, [957].log_data[6].valid := 1, [957].log_data[7].valid := 1, [957].log_data[8].valid := 1, [957].log_data[9].valid := 1, [957].log_data[10].valid := 1, [957].log_data[11].valid := 1, [957].log_data[12].valid := 1, [957].log_data[13].valid := 1, [957].log_data[14].valid := 1, [957].log_data[15].valid := 1, [957].log_data[16].valid := 1, [957].log_data[17].valid := 1, [957].log_data[18].valid := 1, [957].log_data[19].valid := 1, [957].time.Year := 2023, [957].time.Month := 1, [957].time.Day := 13, [957].time.Minute := 9, [957].time.Second := 59, [958].log_data[0].min := 1.0, [958].log_data[0].max := 1.0, [958].log_data[0].total := 300.0, [958].log_data[0].time := 300.0, [958].log_data[0].minminute := 10, [958].log_data[0].maxminute := 10, [958].log_data[0].valid := 1, [958].log_data[1].valid := 1, [958].log_data[2].valid := 1, [958].log_data[3].valid := 1, [958].log_data[4].valid := 1, [958].log_data[5].valid := 1, [958].log_data[6].valid := 1, [958].log_data[7].valid := 1, [958].log_data[8].valid := 1, [958].log_data[9].valid := 1, [958].log_data[10].valid := 1, [958].log_data[11].valid := 1, [958].log_data[12].valid := 1, [958].log_data[13].valid := 1, [958].log_data[14].valid := 1, [958].log_data[15].valid := 1, [958].log_data[16].valid := 1, [958].log_data[17].valid := 1,
        [958].log_data[18].valid := 1, [958].log_data[19].valid := 1, [958].time.Year := 2023, [958].time.Month := 1, [958].time.Day := 13, [958].time.Minute := 14, [958].time.Second := 59, [959].log_data[0].min := 1.0, [959].log_data[0].max := 1.0, [959].log_data[0].total := 300.0, [959].log_data[0].time := 300.0, [959].log_data[0].minminute := 15, [959].log_data[0].maxminute := 15, [959].log_data[0].valid := 1, [959].log_data[1].valid := 1, [959].log_data[2].valid := 1, [959].log_data[3].valid := 1, [959].log_data[4].valid := 1, [959].log_data[5].valid := 1, [959].log_data[6].valid := 1, [959].log_data[7].valid := 1, [959].log_data[8].valid := 1, [959].log_data[9].valid := 1, [959].log_data[10].valid := 1, [959].log_data[11].valid := 1, [959].log_data[12].valid := 1, [959].log_data[13].valid := 1, [959].log_data[14].valid := 1, [959].log_data[15].valid := 1, [959].log_data[16].valid := 1, [959].log_data[17].valid := 1, [959].log_data[18].valid := 1, [959].log_data[19].valid := 1, [959].time.Year := 2023, [959].time.Month := 1, [959].time.Day := 13, [959].time.Minute := 19, [959].time.Second := 59, [960].log_data[0].min := 1.0, [960].log_data[0].max := 1.0, [960].log_data[0].total := 300.0, [960].log_data[0].time := 300.0, [960].log_data[0].minminute := 20, [960].log_data[0].maxminute := 20, [960].log_data[0].valid := 1, [960].log_data[1].valid := 1, [960].log_data[2].valid := 1, [960].log_data[3].valid := 1, [960].log_data[4].valid := 1, [960].log_data[5].valid := 1, [960].log_data[6].valid := 1, [960].log_data[7].valid := 1, [960].log_data[8].valid := 1, [960].log_data[9].valid := 1, [960].log_data[10].valid := 1, [960].log_data[11].valid := 1, [960].log_data[12].valid := 1, [960].log_data[13].valid := 1, [960].log_data[14].valid := 1, [960].log_data[15].valid := 1,
        [960].log_data[16].valid := 1, [960].log_data[17].valid := 1, [960].log_data[18].valid := 1, [960].log_data[19].valid := 1, [960].time.Year := 2023, [960].time.Month := 1, [960].time.Day := 13, [960].time.Minute := 24, [960].time.Second := 59, [961].log_data[0].min := 1.0, [961].log_data[0].max := 1.0, [961].log_data[0].total := 300.0, [961].log_data[0].time := 300.0, [961].log_data[0].minminute := 25, [961].log_data[0].maxminute := 25, [961].log_data[0].valid := 1, [961].log_data[1].valid := 1, [961].log_data[2].valid := 1, [961].log_data[3].valid := 1, [961].log_data[4].valid := 1, [961].log_data[5].valid := 1, [961].log_data[6].valid := 1, [961].log_data[7].valid := 1, [961].log_data[8].valid := 1, [961].log_data[9].valid := 1, [961].log_data[10].valid := 1, [961].log_data[11].valid := 1, [961].log_data[12].valid := 1, [961].log_data[13].valid := 1, [961].log_data[14].valid := 1, [961].log_data[15].valid := 1, [961].log_data[16].valid := 1, [961].log_data[17].valid := 1, [961].log_data[18].valid := 1, [961].log_data[19].valid := 1, [961].time.Year := 2023, [961].time.Month := 1, [961].time.Day := 13, [961].time.Minute := 29, [961].time.Second := 59, [962].log_data[0].min := 1.0, [962].log_data[0].max := 1.0, [962].log_data[0].total := 300.0, [962].log_data[0].time := 300.0, [962].log_data[0].minminute := 30, [962].log_data[0].maxminute := 30, [962].log_data[0].valid := 1, [962].log_data[1].valid := 1, [962].log_data[2].valid := 1, [962].log_data[3].valid := 1, [962].log_data[4].valid := 1, [962].log_data[5].valid := 1, [962].log_data[6].valid := 1, [962].log_data[7].valid := 1, [962].log_data[8].valid := 1, [962].log_data[9].valid := 1, [962].log_data[10].valid := 1, [962].log_data[11].valid := 1, [962].log_data[12].valid := 1, [962].log_data[13].valid := 1,
        [962].log_data[14].valid := 1, [962].log_data[15].valid := 1, [962].log_data[16].valid := 1, [962].log_data[17].valid := 1, [962].log_data[18].valid := 1, [962].log_data[19].valid := 1, [962].time.Year := 2023, [962].time.Month := 1, [962].time.Day := 13, [962].time.Minute := 34, [962].time.Second := 59, [963].log_data[0].min := 1.0, [963].log_data[0].max := 1.0, [963].log_data[0].total := 300.0, [963].log_data[0].time := 300.0, [963].log_data[0].minminute := 35, [963].log_data[0].maxminute := 35, [963].log_data[0].valid := 1, [963].log_data[1].valid := 1, [963].log_data[2].valid := 1, [963].log_data[3].valid := 1, [963].log_data[4].valid := 1, [963].log_data[5].valid := 1, [963].log_data[6].valid := 1, [963].log_data[7].valid := 1, [963].log_data[8].valid := 1, [963].log_data[9].valid := 1, [963].log_data[10].valid := 1, [963].log_data[11].valid := 1, [963].log_data[12].valid := 1, [963].log_data[13].valid := 1, [963].log_data[14].valid := 1, [963].log_data[15].valid := 1, [963].log_data[16].valid := 1, [963].log_data[17].valid := 1, [963].log_data[18].valid := 1, [963].log_data[19].valid := 1, [963].time.Year := 2023, [963].time.Month := 1, [963].time.Day := 13, [963].time.Minute := 39, [963].time.Second := 59, [964].log_data[0].min := 1.0, [964].log_data[0].max := 1.0, [964].log_data[0].total := 300.0, [964].log_data[0].time := 300.0, [964].log_data[0].minminute := 40, [964].log_data[0].maxminute := 40, [964].log_data[0].valid := 1, [964].log_data[1].valid := 1, [964].log_data[2].valid := 1, [964].log_data[3].valid := 1, [964].log_data[4].valid := 1, [964].log_data[5].valid := 1, [964].log_data[6].valid := 1, [964].log_data[7].valid := 1, [964].log_data[8].valid := 1, [964].log_data[9].valid := 1, [964].log_data[10].valid := 1, [964].log_data[11].valid := 1,
        [964].log_data[12].valid := 1, [964].log_data[13].valid := 1, [964].log_data[14].valid := 1, [964].log_data[15].valid := 1, [964].log_data[16].valid := 1, [964].log_data[17].valid := 1, [964].log_data[18].valid := 1, [964].log_data[19].valid := 1, [964].time.Year := 2023, [964].time.Month := 1, [964].time.Day := 13, [964].time.Minute := 44, [964].time.Second := 59, [965].log_data[0].min := 1.0, [965].log_data[0].max := 1.0, [965].log_data[0].total := 300.0, [965].log_data[0].time := 300.0, [965].log_data[0].minminute := 45, [965].log_data[0].maxminute := 45, [965].log_data[0].valid := 1, [965].log_data[1].valid := 1, [965].log_data[2].valid := 1, [965].log_data[3].valid := 1, [965].log_data[4].valid := 1, [965].log_data[5].valid := 1, [965].log_data[6].valid := 1, [965].log_data[7].valid := 1, [965].log_data[8].valid := 1, [965].log_data[9].valid := 1, [965].log_data[10].valid := 1, [965].log_data[11].valid := 1, [965].log_data[12].valid := 1, [965].log_data[13].valid := 1, [965].log_data[14].valid := 1, [965].log_data[15].valid := 1, [965].log_data[16].valid := 1, [965].log_data[17].valid := 1, [965].log_data[18].valid := 1, [965].log_data[19].valid := 1, [965].time.Year := 2023, [965].time.Month := 1, [965].time.Day := 13, [965].time.Minute := 49, [965].time.Second := 59, [966].log_data[0].min := 1.0, [966].log_data[0].max := 1.0, [966].log_data[0].total := 300.0, [966].log_data[0].time := 300.0, [966].log_data[0].minminute := 50, [966].log_data[0].maxminute := 50, [966].log_data[0].valid := 1, [966].log_data[1].valid := 1, [966].log_data[2].valid := 1, [966].log_data[3].valid := 1, [966].log_data[4].valid := 1, [966].log_data[5].valid := 1, [966].log_data[6].valid := 1, [966].log_data[7].valid := 1, [966].log_data[8].valid := 1, [966].log_data[9].valid := 1,
        [966].log_data[10].valid := 1, [966].log_data[11].valid := 1, [966].log_data[12].valid := 1, [966].log_data[13].valid := 1, [966].log_data[14].valid := 1, [966].log_data[15].valid := 1, [966].log_data[16].valid := 1, [966].log_data[17].valid := 1, [966].log_data[18].valid := 1, [966].log_data[19].valid := 1, [966].time.Year := 2023, [966].time.Month := 1, [966].time.Day := 13, [966].time.Minute := 54, [966].time.Second := 59, [967].log_data[0].min := 1.0, [967].log_data[0].max := 1.0, [967].log_data[0].total := 300.0, [967].log_data[0].time := 300.0, [967].log_data[0].minminute := 55, [967].log_data[0].maxminute := 55, [967].log_data[0].valid := 1, [967].log_data[1].valid := 1, [967].log_data[2].valid := 1, [967].log_data[3].valid := 1, [967].log_data[4].valid := 1, [967].log_data[5].valid := 1, [967].log_data[6].valid := 1, [967].log_data[7].valid := 1, [967].log_data[8].valid := 1, [967].log_data[9].valid := 1, [967].log_data[10].valid := 1, [967].log_data[11].valid := 1, [967].log_data[12].valid := 1, [967].log_data[13].valid := 1, [967].log_data[14].valid := 1, [967].log_data[15].valid := 1, [967].log_data[16].valid := 1, [967].log_data[17].valid := 1, [967].log_data[18].valid := 1, [967].log_data[19].valid := 1, [967].time.Year := 2023, [967].time.Month := 1, [967].time.Day := 13, [967].time.Minute := 59, [967].time.Second := 59, [968].log_data[0].min := 1.0, [968].log_data[0].max := 1.0, [968].log_data[0].total := 299.5, [968].log_data[0].time := 299.5, [968].log_data[0].valid := 1, [968].log_data[1].valid := 1, [968].log_data[2].valid := 1, [968].log_data[3].valid := 1, [968].log_data[4].valid := 1, [968].log_data[5].valid := 1, [968].log_data[6].valid := 1, [968].log_data[7].valid := 1, [968].log_data[8].valid := 1, [968].log_data[9].valid := 1,
        [968].log_data[10].valid := 1, [968].log_data[11].valid := 1, [968].log_data[12].valid := 1, [968].log_data[13].valid := 1, [968].log_data[14].valid := 1, [968].log_data[15].valid := 1, [968].log_data[16].valid := 1, [968].log_data[17].valid := 1, [968].log_data[18].valid := 1, [968].log_data[19].valid := 1, [968].time.Year := 2023, [968].time.Month := 1, [968].time.Day := 13, [968].time.Hour := 1, [968].time.Minute := 4, [968].time.Second := 59, [969].log_data[0].min := 1.0, [969].log_data[0].max := 1.0, [969].log_data[0].total := 300.0, [969].log_data[0].time := 300.0, [969].log_data[0].minminute := 5, [969].log_data[0].maxminute := 5, [969].log_data[0].valid := 1, [969].log_data[1].valid := 1, [969].log_data[2].valid := 1, [969].log_data[3].valid := 1, [969].log_data[4].valid := 1, [969].log_data[5].valid := 1, [969].log_data[6].valid := 1, [969].log_data[7].valid := 1, [969].log_data[8].valid := 1, [969].log_data[9].valid := 1, [969].log_data[10].valid := 1, [969].log_data[11].valid := 1, [969].log_data[12].valid := 1, [969].log_data[13].valid := 1, [969].log_data[14].valid := 1, [969].log_data[15].valid := 1, [969].log_data[16].valid := 1, [969].log_data[17].valid := 1, [969].log_data[18].valid := 1, [969].log_data[19].valid := 1, [969].time.Year := 2023, [969].time.Month := 1, [969].time.Day := 13, [969].time.Hour := 1, [969].time.Minute := 9, [969].time.Second := 59, [970].log_data[0].min := 1.0, [970].log_data[0].max := 1.0, [970].log_data[0].total := 300.0, [970].log_data[0].time := 300.0, [970].log_data[0].minminute := 10, [970].log_data[0].maxminute := 10, [970].log_data[0].valid := 1, [970].log_data[1].valid := 1, [970].log_data[2].valid := 1, [970].log_data[3].valid := 1, [970].log_data[4].valid := 1, [970].log_data[5].valid := 1,
        [970].log_data[6].valid := 1, [970].log_data[7].valid := 1, [970].log_data[8].valid := 1, [970].log_data[9].valid := 1, [970].log_data[10].valid := 1, [970].log_data[11].valid := 1, [970].log_data[12].valid := 1, [970].log_data[13].valid := 1, [970].log_data[14].valid := 1, [970].log_data[15].valid := 1, [970].log_data[16].valid := 1, [970].log_data[17].valid := 1, [970].log_data[18].valid := 1, [970].log_data[19].valid := 1, [970].time.Year := 2023, [970].time.Month := 1, [970].time.Day := 13, [970].time.Hour := 1, [970].time.Minute := 14, [970].time.Second := 59, [971].log_data[0].min := 1.0, [971].log_data[0].max := 1.0, [971].log_data[0].total := 300.0, [971].log_data[0].time := 300.0, [971].log_data[0].minminute := 15, [971].log_data[0].maxminute := 15, [971].log_data[0].valid := 1, [971].log_data[1].valid := 1, [971].log_data[2].valid := 1, [971].log_data[3].valid := 1, [971].log_data[4].valid := 1, [971].log_data[5].valid := 1, [971].log_data[6].valid := 1, [971].log_data[7].valid := 1, [971].log_data[8].valid := 1, [971].log_data[9].valid := 1, [971].log_data[10].valid := 1, [971].log_data[11].valid := 1, [971].log_data[12].valid := 1, [971].log_data[13].valid := 1, [971].log_data[14].valid := 1, [971].log_data[15].valid := 1, [971].log_data[16].valid := 1, [971].log_data[17].valid := 1, [971].log_data[18].valid := 1, [971].log_data[19].valid := 1, [971].time.Year := 2023, [971].time.Month := 1, [971].time.Day := 13, [971].time.Hour := 1, [971].time.Minute := 19, [971].time.Second := 59, [972].log_data[0].min := 1.0, [972].log_data[0].max := 1.0, [972].log_data[0].total := 300.0, [972].log_data[0].time := 300.0, [972].log_data[0].minminute := 20, [972].log_data[0].maxminute := 20, [972].log_data[0].valid := 1, [972].log_data[1].valid := 1,
        [972].log_data[2].valid := 1, [972].log_data[3].valid := 1, [972].log_data[4].valid := 1, [972].log_data[5].valid := 1, [972].log_data[6].valid := 1, [972].log_data[7].valid := 1, [972].log_data[8].valid := 1, [972].log_data[9].valid := 1, [972].log_data[10].valid := 1, [972].log_data[11].valid := 1, [972].log_data[12].valid := 1, [972].log_data[13].valid := 1, [972].log_data[14].valid := 1, [972].log_data[15].valid := 1, [972].log_data[16].valid := 1, [972].log_data[17].valid := 1, [972].log_data[18].valid := 1, [972].log_data[19].valid := 1, [972].time.Year := 2023, [972].time.Month := 1, [972].time.Day := 13, [972].time.Hour := 1, [972].time.Minute := 24, [972].time.Second := 59, [973].log_data[0].min := 1.0, [973].log_data[0].max := 1.0, [973].log_data[0].total := 300.0, [973].log_data[0].time := 300.0, [973].log_data[0].minminute := 25, [973].log_data[0].maxminute := 25, [973].log_data[0].valid := 1, [973].log_data[1].valid := 1, [973].log_data[2].valid := 1, [973].log_data[3].valid := 1, [973].log_data[4].valid := 1, [973].log_data[5].valid := 1, [973].log_data[6].valid := 1, [973].log_data[7].valid := 1, [973].log_data[8].valid := 1, [973].log_data[9].valid := 1, [973].log_data[10].valid := 1, [973].log_data[11].valid := 1, [973].log_data[12].valid := 1, [973].log_data[13].valid := 1, [973].log_data[14].valid := 1, [973].log_data[15].valid := 1, [973].log_data[16].valid := 1, [973].log_data[17].valid := 1, [973].log_data[18].valid := 1, [973].log_data[19].valid := 1, [973].time.Year := 2023, [973].time.Month := 1, [973].time.Day := 13, [973].time.Hour := 1, [973].time.Minute := 29, [973].time.Second := 59, [974].log_data[0].min := 1.0, [974].log_data[0].max := 1.0, [974].log_data[0].total := 300.0, [974].log_data[0].time := 300.0,
        [974].log_data[0].minminute := 30, [974].log_data[0].maxminute := 30, [974].log_data[0].valid := 1, [974].log_data[1].valid := 1, [974].log_data[2].valid := 1, [974].log_data[3].valid := 1, [974].log_data[4].valid := 1, [974].log_data[5].valid := 1, [974].log_data[6].valid := 1, [974].log_data[7].valid := 1, [974].log_data[8].valid := 1, [974].log_data[9].valid := 1, [974].log_data[10].valid := 1, [974].log_data[11].valid := 1, [974].log_data[12].valid := 1, [974].log_data[13].valid := 1, [974].log_data[14].valid := 1, [974].log_data[15].valid := 1, [974].log_data[16].valid := 1, [974].log_data[17].valid := 1, [974].log_data[18].valid := 1, [974].log_data[19].valid := 1, [974].time.Year := 2023, [974].time.Month := 1, [974].time.Day := 13, [974].time.Hour := 1, [974].time.Minute := 34, [974].time.Second := 59, [975].log_data[0].min := 1.0, [975].log_data[0].max := 1.0, [975].log_data[0].total := 300.0, [975].log_data[0].time := 300.0, [975].log_data[0].minminute := 35, [975].log_data[0].maxminute := 35, [975].log_data[0].valid := 1, [975].log_data[1].valid := 1, [975].log_data[2].valid := 1, [975].log_data[3].valid := 1, [975].log_data[4].valid := 1, [975].log_data[5].valid := 1, [975].log_data[6].valid := 1, [975].log_data[7].valid := 1, [975].log_data[8].valid := 1, [975].log_data[9].valid := 1, [975].log_data[10].valid := 1, [975].log_data[11].valid := 1, [975].log_data[12].valid := 1, [975].log_data[13].valid := 1, [975].log_data[14].valid := 1, [975].log_data[15].valid := 1, [975].log_data[16].valid := 1, [975].log_data[17].valid := 1, [975].log_data[18].valid := 1, [975].log_data[19].valid := 1, [975].time.Year := 2023, [975].time.Month := 1, [975].time.Day := 13, [975].time.Hour := 1, [975].time.Minute := 39, [975].time.Second := 59,
        [976].log_data[0].min := 1.0, [976].log_data[0].max := 1.0, [976].log_data[0].total := 300.0, [976].log_data[0].time := 300.0, [976].log_data[0].minminute := 40, [976].log_data[0].maxminute := 40, [976].log_data[0].valid := 1, [976].log_data[1].valid := 1, [976].log_data[2].valid := 1, [976].log_data[3].valid := 1, [976].log_data[4].valid := 1, [976].log_data[5].valid := 1, [976].log_data[6].valid := 1, [976].log_data[7].valid := 1, [976].log_data[8].valid := 1, [976].log_data[9].valid := 1, [976].log_data[10].valid := 1, [976].log_data[11].valid := 1, [976].log_data[12].valid := 1, [976].log_data[13].valid := 1, [976].log_data[14].valid := 1, [976].log_data[15].valid := 1, [976].log_data[16].valid := 1, [976].log_data[17].valid := 1, [976].log_data[18].valid := 1, [976].log_data[19].valid := 1, [976].time.Year := 2023, [976].time.Month := 1, [976].time.Day := 13, [976].time.Hour := 1, [976].time.Minute := 44, [976].time.Second := 59, [977].log_data[0].min := 1.0, [977].log_data[0].max := 1.0, [977].log_data[0].total := 300.0, [977].log_data[0].time := 300.0, [977].log_data[0].minminute := 45, [977].log_data[0].maxminute := 45, [977].log_data[0].valid := 1, [977].log_data[1].valid := 1, [977].log_data[2].valid := 1, [977].log_data[3].valid := 1, [977].log_data[4].valid := 1, [977].log_data[5].valid := 1, [977].log_data[6].valid := 1, [977].log_data[7].valid := 1, [977].log_data[8].valid := 1, [977].log_data[9].valid := 1, [977].log_data[10].valid := 1, [977].log_data[11].valid := 1, [977].log_data[12].valid := 1, [977].log_data[13].valid := 1, [977].log_data[14].valid := 1, [977].log_data[15].valid := 1, [977].log_data[16].valid := 1, [977].log_data[17].valid := 1, [977].log_data[18].valid := 1, [977].log_data[19].valid := 1, [977].time.Year := 2023, [977].time.Month := 1,
        [977].time.Day := 13, [977].time.Hour := 1, [977].time.Minute := 49, [977].time.Second := 59, [978].log_data[0].min := 1.0, [978].log_data[0].max := 1.0, [978].log_data[0].total := 300.0, [978].log_data[0].time := 300.0, [978].log_data[0].minminute := 50, [978].log_data[0].maxminute := 50, [978].log_data[0].valid := 1, [978].log_data[1].valid := 1, [978].log_data[2].valid := 1, [978].log_data[3].valid := 1, [978].log_data[4].valid := 1, [978].log_data[5].valid := 1, [978].log_data[6].valid := 1, [978].log_data[7].valid := 1, [978].log_data[8].valid := 1, [978].log_data[9].valid := 1, [978].log_data[10].valid := 1, [978].log_data[11].valid := 1, [978].log_data[12].valid := 1, [978].log_data[13].valid := 1, [978].log_data[14].valid := 1, [978].log_data[15].valid := 1, [978].log_data[16].valid := 1, [978].log_data[17].valid := 1, [978].log_data[18].valid := 1, [978].log_data[19].valid := 1, [978].time.Year := 2023, [978].time.Month := 1, [978].time.Day := 13, [978].time.Hour := 1, [978].time.Minute := 54, [978].time.Second := 59, [979].log_data[0].min := 1.0, [979].log_data[0].max := 1.0, [979].log_data[0].total := 300.0, [979].log_data[0].time := 300.0, [979].log_data[0].minminute := 55, [979].log_data[0].maxminute := 55, [979].log_data[0].valid := 1, [979].log_data[1].valid := 1, [979].log_data[2].valid := 1, [979].log_data[3].valid := 1, [979].log_data[4].valid := 1, [979].log_data[5].valid := 1, [979].log_data[6].valid := 1, [979].log_data[7].valid := 1, [979].log_data[8].valid := 1, [979].log_data[9].valid := 1, [979].log_data[10].valid := 1, [979].log_data[11].valid := 1, [979].log_data[12].valid := 1, [979].log_data[13].valid := 1, [979].log_data[14].valid := 1, [979].log_data[15].valid := 1, [979].log_data[16].valid := 1, [979].log_data[17].valid := 1,
        [979].log_data[18].valid := 1, [979].log_data[19].valid := 1, [979].time.Year := 2023, [979].time.Month := 1, [979].time.Day := 13, [979].time.Hour := 1, [979].time.Minute := 59, [979].time.Second := 59, [980].log_data[0].min := 1.0, [980].log_data[0].max := 1.0, [980].log_data[0].total := 300.0, [980].log_data[0].time := 300.0, [980].log_data[0].valid := 1, [980].log_data[1].valid := 1, [980].log_data[2].valid := 1, [980].log_data[3].valid := 1, [980].log_data[4].valid := 1, [980].log_data[5].valid := 1, [980].log_data[6].valid := 1, [980].log_data[7].valid := 1, [980].log_data[8].valid := 1, [980].log_data[9].valid := 1, [980].log_data[10].valid := 1, [980].log_data[11].valid := 1, [980].log_data[12].valid := 1, [980].log_data[13].valid := 1, [980].log_data[14].valid := 1, [980].log_data[15].valid := 1, [980].log_data[16].valid := 1, [980].log_data[17].valid := 1, [980].log_data[18].valid := 1, [980].log_data[19].valid := 1, [980].time.Year := 2023, [980].time.Month := 1, [980].time.Day := 13, [980].time.Hour := 2, [980].time.Minute := 4, [980].time.Second := 59, [981].log_data[0].min := 1.0, [981].log_data[0].max := 1.0, [981].log_data[0].total := 300.0, [981].log_data[0].time := 300.0, [981].log_data[0].minminute := 5, [981].log_data[0].maxminute := 5, [981].log_data[0].valid := 1, [981].log_data[1].valid := 1, [981].log_data[2].valid := 1, [981].log_data[3].valid := 1, [981].log_data[4].valid := 1, [981].log_data[5].valid := 1, [981].log_data[6].valid := 1, [981].log_data[7].valid := 1, [981].log_data[8].valid := 1, [981].log_data[9].valid := 1, [981].log_data[10].valid := 1, [981].log_data[11].valid := 1, [981].log_data[12].valid := 1, [981].log_data[13].valid := 1, [981].log_data[14].valid := 1, [981].log_data[15].valid := 1,
        [981].log_data[16].valid := 1, [981].log_data[17].valid := 1, [981].log_data[18].valid := 1, [981].log_data[19].valid := 1, [981].time.Year := 2023, [981].time.Month := 1, [981].time.Day := 13, [981].time.Hour := 2, [981].time.Minute := 9, [981].time.Second := 59, [982].log_data[0].min := 1.0, [982].log_data[0].max := 1.0, [982].log_data[0].total := 300.0, [982].log_data[0].time := 300.0, [982].log_data[0].minminute := 10, [982].log_data[0].maxminute := 10, [982].log_data[0].valid := 1, [982].log_data[1].valid := 1, [982].log_data[2].valid := 1, [982].log_data[3].valid := 1, [982].log_data[4].valid := 1, [982].log_data[5].valid := 1, [982].log_data[6].valid := 1, [982].log_data[7].valid := 1, [982].log_data[8].valid := 1, [982].log_data[9].valid := 1, [982].log_data[10].valid := 1, [982].log_data[11].valid := 1, [982].log_data[12].valid := 1, [982].log_data[13].valid := 1, [982].log_data[14].valid := 1, [982].log_data[15].valid := 1, [982].log_data[16].valid := 1, [982].log_data[17].valid := 1, [982].log_data[18].valid := 1, [982].log_data[19].valid := 1, [982].time.Year := 2023, [982].time.Month := 1, [982].time.Day := 13, [982].time.Hour := 2, [982].time.Minute := 14, [982].time.Second := 59, [983].log_data[0].min := 1.0, [983].log_data[0].max := 1.0, [983].log_data[0].total := 300.0, [983].log_data[0].time := 300.0, [983].log_data[0].minminute := 15, [983].log_data[0].maxminute := 15, [983].log_data[0].valid := 1, [983].log_data[1].valid := 1, [983].log_data[2].valid := 1, [983].log_data[3].valid := 1, [983].log_data[4].valid := 1, [983].log_data[5].valid := 1, [983].log_data[6].valid := 1, [983].log_data[7].valid := 1, [983].log_data[8].valid := 1, [983].log_data[9].valid := 1, [983].log_data[10].valid := 1, [983].log_data[11].valid := 1,
        [983].log_data[12].valid := 1, [983].log_data[13].valid := 1, [983].log_data[14].valid := 1, [983].log_data[15].valid := 1, [983].log_data[16].valid := 1, [983].log_data[17].valid := 1, [983].log_data[18].valid := 1, [983].log_data[19].valid := 1, [983].time.Year := 2023, [983].time.Month := 1, [983].time.Day := 13, [983].time.Hour := 2, [983].time.Minute := 19, [983].time.Second := 59, [984].log_data[0].min := 1.0, [984].log_data[0].max := 1.0, [984].log_data[0].total := 300.0, [984].log_data[0].time := 300.0, [984].log_data[0].minminute := 20, [984].log_data[0].maxminute := 20, [984].log_data[0].valid := 1, [984].log_data[1].valid := 1, [984].log_data[2].valid := 1, [984].log_data[3].valid := 1, [984].log_data[4].valid := 1, [984].log_data[5].valid := 1, [984].log_data[6].valid := 1, [984].log_data[7].valid := 1, [984].log_data[8].valid := 1, [984].log_data[9].valid := 1, [984].log_data[10].valid := 1, [984].log_data[11].valid := 1, [984].log_data[12].valid := 1, [984].log_data[13].valid := 1, [984].log_data[14].valid := 1, [984].log_data[15].valid := 1, [984].log_data[16].valid := 1, [984].log_data[17].valid := 1, [984].log_data[18].valid := 1, [984].log_data[19].valid := 1, [984].time.Year := 2023, [984].time.Month := 1, [984].time.Day := 13, [984].time.Hour := 2, [984].time.Minute := 24, [984].time.Second := 59, [985].log_data[0].min := 1.0, [985].log_data[0].max := 1.0, [985].log_data[0].total := 300.0, [985].log_data[0].time := 300.0, [985].log_data[0].minminute := 25, [985].log_data[0].maxminute := 25, [985].log_data[0].valid := 1, [985].log_data[1].valid := 1, [985].log_data[2].valid := 1, [985].log_data[3].valid := 1, [985].log_data[4].valid := 1, [985].log_data[5].valid := 1, [985].log_data[6].valid := 1, [985].log_data[7].valid := 1,
        [985].log_data[8].valid := 1, [985].log_data[9].valid := 1, [985].log_data[10].valid := 1, [985].log_data[11].valid := 1, [985].log_data[12].valid := 1, [985].log_data[13].valid := 1, [985].log_data[14].valid := 1, [985].log_data[15].valid := 1, [985].log_data[16].valid := 1, [985].log_data[17].valid := 1, [985].log_data[18].valid := 1, [985].log_data[19].valid := 1, [985].time.Year := 2023, [985].time.Month := 1, [985].time.Day := 13, [985].time.Hour := 2, [985].time.Minute := 29, [985].time.Second := 59, [986].log_data[0].min := 1.0, [986].log_data[0].max := 1.0, [986].log_data[0].total := 300.0, [986].log_data[0].time := 300.0, [986].log_data[0].minminute := 30, [986].log_data[0].maxminute := 30, [986].log_data[0].valid := 1, [986].log_data[1].valid := 1, [986].log_data[2].valid := 1, [986].log_data[3].valid := 1, [986].log_data[4].valid := 1, [986].log_data[5].valid := 1, [986].log_data[6].valid := 1, [986].log_data[7].valid := 1, [986].log_data[8].valid := 1, [986].log_data[9].valid := 1, [986].log_data[10].valid := 1, [986].log_data[11].valid := 1, [986].log_data[12].valid := 1, [986].log_data[13].valid := 1, [986].log_data[14].valid := 1, [986].log_data[15].valid := 1, [986].log_data[16].valid := 1, [986].log_data[17].valid := 1, [986].log_data[18].valid := 1, [986].log_data[19].valid := 1, [986].time.Year := 2023, [986].time.Month := 1, [986].time.Day := 13, [986].time.Hour := 2, [986].time.Minute := 34, [986].time.Second := 59, [987].log_data[0].min := 1.0, [987].log_data[0].max := 1.0, [987].log_data[0].total := 300.0, [987].log_data[0].time := 300.0, [987].log_data[0].minminute := 35, [987].log_data[0].maxminute := 35, [987].log_data[0].valid := 1, [987].log_data[1].valid := 1, [987].log_data[2].valid := 1, [987].log_data[3].valid := 1,
        [987].log_data[4].valid := 1, [987].log_data[5].valid := 1, [987].log_data[6].valid := 1, [987].log_data[7].valid := 1, [987].log_data[8].valid := 1, [987].log_data[9].valid := 1, [987].log_data[10].valid := 1, [987].log_data[11].valid := 1, [987].log_data[12].valid := 1, [987].log_data[13].valid := 1, [987].log_data[14].valid := 1, [987].log_data[15].valid := 1, [987].log_data[16].valid := 1, [987].log_data[17].valid := 1, [987].log_data[18].valid := 1, [987].log_data[19].valid := 1, [987].time.Year := 2023, [987].time.Month := 1, [987].time.Day := 13, [987].time.Hour := 2, [987].time.Minute := 39, [987].time.Second := 59, [988].log_data[0].min := 1.0, [988].log_data[0].max := 1.0, [988].log_data[0].total := 300.0, [988].log_data[0].time := 300.0, [988].log_data[0].minminute := 40, [988].log_data[0].maxminute := 40, [988].log_data[0].valid := 1, [988].log_data[1].valid := 1, [988].log_data[2].valid := 1, [988].log_data[3].valid := 1, [988].log_data[4].valid := 1, [988].log_data[5].valid := 1, [988].log_data[6].valid := 1, [988].log_data[7].valid := 1, [988].log_data[8].valid := 1, [988].log_data[9].valid := 1, [988].log_data[10].valid := 1, [988].log_data[11].valid := 1, [988].log_data[12].valid := 1, [988].log_data[13].valid := 1, [988].log_data[14].valid := 1, [988].log_data[15].valid := 1, [988].log_data[16].valid := 1, [988].log_data[17].valid := 1, [988].log_data[18].valid := 1, [988].log_data[19].valid := 1, [988].time.Year := 2023, [988].time.Month := 1, [988].time.Day := 13, [988].time.Hour := 2, [988].time.Minute := 44, [988].time.Second := 59, [989].log_data[0].min := 1.0, [989].log_data[0].max := 1.0, [989].log_data[0].total := 300.0, [989].log_data[0].time := 300.0, [989].log_data[0].minminute := 45, [989].log_data[0].maxminute := 45,
        [989].log_data[0].valid := 1, [989].log_data[1].valid := 1, [989].log_data[2].valid := 1, [989].log_data[3].valid := 1, [989].log_data[4].valid := 1, [989].log_data[5].valid := 1, [989].log_data[6].valid := 1, [989].log_data[7].valid := 1, [989].log_data[8].valid := 1, [989].log_data[9].valid := 1, [989].log_data[10].valid := 1, [989].log_data[11].valid := 1, [989].log_data[12].valid := 1, [989].log_data[13].valid := 1, [989].log_data[14].valid := 1, [989].log_data[15].valid := 1, [989].log_data[16].valid := 1, [989].log_data[17].valid := 1, [989].log_data[18].valid := 1, [989].log_data[19].valid := 1, [989].time.Year := 2023, [989].time.Month := 1, [989].time.Day := 13, [989].time.Hour := 2, [989].time.Minute := 49, [989].time.Second := 59, [990].log_data[0].min := 1.0, [990].log_data[0].max := 1.0, [990].log_data[0].total := 300.0, [990].log_data[0].time := 300.0, [990].log_data[0].minminute := 50, [990].log_data[0].maxminute := 50, [990].log_data[0].valid := 1, [990].log_data[1].valid := 1, [990].log_data[2].valid := 1, [990].log_data[3].valid := 1, [990].log_data[4].valid := 1, [990].log_data[5].valid := 1, [990].log_data[6].valid := 1, [990].log_data[7].valid := 1, [990].log_data[8].valid := 1, [990].log_data[9].valid := 1, [990].log_data[10].valid := 1, [990].log_data[11].valid := 1, [990].log_data[12].valid := 1, [990].log_data[13].valid := 1, [990].log_data[14].valid := 1, [990].log_data[15].valid := 1, [990].log_data[16].valid := 1, [990].log_data[17].valid := 1, [990].log_data[18].valid := 1, [990].log_data[19].valid := 1, [990].time.Year := 2023, [990].time.Month := 1, [990].time.Day := 13, [990].time.Hour := 2, [990].time.Minute := 54, [990].time.Second := 59, [991].log_data[0].min := 1.0, [991].log_data[0].max := 1.0,
        [991].log_data[0].total := 300.0, [991].log_data[0].time := 300.0, [991].log_data[0].minminute := 55, [991].log_data[0].maxminute := 55, [991].log_data[0].valid := 1, [991].log_data[1].valid := 1, [991].log_data[2].valid := 1, [991].log_data[3].valid := 1, [991].log_data[4].valid := 1, [991].log_data[5].valid := 1, [991].log_data[6].valid := 1, [991].log_data[7].valid := 1, [991].log_data[8].valid := 1, [991].log_data[9].valid := 1, [991].log_data[10].valid := 1, [991].log_data[11].valid := 1, [991].log_data[12].valid := 1, [991].log_data[13].valid := 1, [991].log_data[14].valid := 1, [991].log_data[15].valid := 1, [991].log_data[16].valid := 1, [991].log_data[17].valid := 1, [991].log_data[18].valid := 1, [991].log_data[19].valid := 1, [991].time.Year := 2023, [991].time.Month := 1, [991].time.Day := 13, [991].time.Hour := 2, [991].time.Minute := 59, [991].time.Second := 59, [992].log_data[0].min := 1.0, [992].log_data[0].max := 1.0, [992].log_data[0].total := 300.0, [992].log_data[0].time := 300.0, [992].log_data[0].valid := 1, [992].log_data[1].valid := 1, [992].log_data[2].valid := 1, [992].log_data[3].valid := 1, [992].log_data[4].valid := 1, [992].log_data[5].valid := 1, [992].log_data[6].valid := 1, [992].log_data[7].valid := 1, [992].log_data[8].valid := 1, [992].log_data[9].valid := 1, [992].log_data[10].valid := 1, [992].log_data[11].valid := 1, [992].log_data[12].valid := 1, [992].log_data[13].valid := 1, [992].log_data[14].valid := 1, [992].log_data[15].valid := 1, [992].log_data[16].valid := 1, [992].log_data[17].valid := 1, [992].log_data[18].valid := 1, [992].log_data[19].valid := 1, [992].time.Year := 2023, [992].time.Month := 1, [992].time.Day := 13, [992].time.Hour := 3, [992].time.Minute := 4, [992].time.Second := 59,
        [993].log_data[0].min := 1.0, [993].log_data[0].max := 1.0, [993].log_data[0].total := 300.0, [993].log_data[0].time := 300.0, [993].log_data[0].minminute := 5, [993].log_data[0].maxminute := 5, [993].log_data[0].valid := 1, [993].log_data[1].valid := 1, [993].log_data[2].valid := 1, [993].log_data[3].valid := 1, [993].log_data[4].valid := 1, [993].log_data[5].valid := 1, [993].log_data[6].valid := 1, [993].log_data[7].valid := 1, [993].log_data[8].valid := 1, [993].log_data[9].valid := 1, [993].log_data[10].valid := 1, [993].log_data[11].valid := 1, [993].log_data[12].valid := 1, [993].log_data[13].valid := 1, [993].log_data[14].valid := 1, [993].log_data[15].valid := 1, [993].log_data[16].valid := 1, [993].log_data[17].valid := 1, [993].log_data[18].valid := 1, [993].log_data[19].valid := 1, [993].time.Year := 2023, [993].time.Month := 1, [993].time.Day := 13, [993].time.Hour := 3, [993].time.Minute := 9, [993].time.Second := 59, [994].log_data[0].min := 1.0, [994].log_data[0].max := 1.0, [994].log_data[0].total := 300.0, [994].log_data[0].time := 300.0, [994].log_data[0].minminute := 10, [994].log_data[0].maxminute := 10, [994].log_data[0].valid := 1, [994].log_data[1].valid := 1, [994].log_data[2].valid := 1, [994].log_data[3].valid := 1, [994].log_data[4].valid := 1, [994].log_data[5].valid := 1, [994].log_data[6].valid := 1, [994].log_data[7].valid := 1, [994].log_data[8].valid := 1, [994].log_data[9].valid := 1, [994].log_data[10].valid := 1, [994].log_data[11].valid := 1, [994].log_data[12].valid := 1, [994].log_data[13].valid := 1, [994].log_data[14].valid := 1, [994].log_data[15].valid := 1, [994].log_data[16].valid := 1, [994].log_data[17].valid := 1, [994].log_data[18].valid := 1, [994].log_data[19].valid := 1, [994].time.Year := 2023, [994].time.Month := 1,
